LIN {X 0,Y 187.273,Z 370.418,A -85,B 0,C 180,E1 -25349.144,E2 -25349.144} C_VEL
LIN {X 0,Y 191.454,Z 356.11,A -85,B 0,C 180,E1 -25350.14,E2 -25350.14} C_VEL
LIN {X 0,Y 194.75,Z 340.819,A -85,B 0,C 180,E1 -25350.906,E2 -25350.906} C_VEL
LIN {X 0,Y 196.826,Z 325.628,A -85,B 0,C 180,E1 -25351.428,E2 -25351.428} C_VEL
LIN {X 0,Y 201.138,Z 277.904,A -85,B 0,C 180,E1 -25352.703,E2 -25352.703} C_VEL
LIN {X 0,Y 197.64,Z 268.624,A -85,B 0,C 180,E1 -25355.513,E2 -25355.513} C_VEL
LIN {X 0,Y 193.851,Z 261.276,A -85,B 0,C 180,E1 -25358.813,E2 -25358.813} C_VEL
LIN {X 0,Y 190.051,Z 254.613,A -85,B 0,C 180,E1 -25362.793,E2 -25362.793} C_VEL
LIN {X 0,Y 187.566,Z 250.534,A -85,B 0,C 180,E1 -25366.042,E2 -25366.042} C_VEL
LIN {X 0,Y 185.493,Z 246.833,A -85,B 0,C 180,E1 -25369.632,E2 -25369.632} C_VEL
LIN {X 0,Y 183.537,Z 243.434,A -85,B 0,C 180,E1 -25375.058,E2 -25375.058} C_VEL
LIN {X 0,Y 183.272,Z 242.439,A -85,B 0,C 180,E1 -25376.703,E2 -25376.703} C_VEL
LIN {X 0,Y 183.007,Z 241.999,A -85,B 0,C 180,E1 -25380,E2 -25380} C_VEL
LIN {X 0,Y 183.335,Z 242.534,A -85,B 0,C 180,E1 -25383.847,E2 -25383.847} C_VEL
LIN {X 0,Y 184.872,Z 246.218,A -85,B 0,C 180,E1 -25389.298,E2 -25389.298} C_VEL
LIN {X 0,Y 185.731,Z 247.38,A -85,B 0,C 180,E1 -25391.044,E2 -25391.044} C_VEL
LIN {X 0,Y 188.365,Z 251.957,A -85,B 0,C 180,E1 -25395.278,E2 -25395.278} C_VEL
LIN {X 0,Y 190.886,Z 256.242,A -85,B 0,C 180,E1 -25398.364,E2 -25398.364} C_VEL
LIN {X 0,Y 193.99,Z 261.588,A -85,B 0,C 180,E1 -25401.5,E2 -25401.5} C_VEL
LIN {X 0,Y 198.275,Z 269.947,A -85,B 0,C 180,E1 -25405.173,E2 -25405.173} C_VEL
LIN {X 0,Y 201.262,Z 276.327,A -85,B 0,C 180,E1 -25407.421,E2 -25407.421} C_VEL
LIN {X 0,Y 196.205,Z 330.798,A -85,B 0,C 180,E1 -25408.917,E2 -25408.917} C_VEL
LIN {X 0,Y 193.603,Z 345.867,A -85,B 0,C 180,E1 -25409.531,E2 -25409.531} C_VEL
LIN {X 0,Y 189.657,Z 361.736,A -85,B 0,C 180,E1 -25410.507,E2 -25410.507} C_VEL
LIN {X 0,Y 185.585,Z 374.397,A -85,B 0,C 180,E1 -25411.563,E2 -25411.563} C_VEL
LIN {X 0,Y 180.029,Z 388.733,A -85,B 0,C 180,E1 -25413.184,E2 -25413.184} C_VEL
LIN {X 0,Y 173.921,Z 401.727,A -85,B 0,C 180,E1 -25415.087,E2 -25415.087} C_VEL
LIN {X 0,Y 167.017,Z 414.16,A -85,B 0,C 180,E1 -25417.415,E2 -25417.415} C_VEL
LIN {X 0,Y 160.472,Z 424.572,A -85,B 0,C 180,E1 -25419.966,E2 -25419.966} C_VEL
LIN {X 0,Y 153.641,Z 434.234,A -85,B 0,C 180,E1 -25422.955,E2 -25422.955} C_VEL
LIN {X 0,Y 147.458,Z 442.478,A -85,B 0,C 180,E1 -25426.284,E2 -25426.284} C_VEL
LIN {X 0,Y 140.675,Z 450.588,A -85,B 0,C 180,E1 -25430.433,E2 -25430.433} C_VEL
LIN {X 0,Y 134.787,Z 457.281,A -85,B 0,C 180,E1 -25435.001,E2 -25435.001} C_VEL
LIN {X 0,Y 129.035,Z 463.475,A -85,B 0,C 180,E1 -25440.647,E2 -25440.647} C_VEL
LIN {X 0,Y 124.739,Z 468.254,A -85,B 0,C 180,E1 -25446.772,E2 -25446.772} C_VEL
LIN {X 0,Y 121.613,Z 471.753,A -85,B 0,C 180,E1 -25453.205,E2 -25453.205} C_VEL
LIN {X 0,Y 119.848,Z 474.061,A -85,B 0,C 180,E1 -25459.868,E2 -25459.868} C_VEL
LIN {X 0,Y 119.226,Z 475.233,A -85,B 0,C 180,E1 -25466.621,E2 -25466.621} C_VEL
LIN {X 0,Y 119.279,Z 475.389,A -85,B 0,C 180,E1 -25470,E2 -25470} C_VEL
LIN {X 0,Y 119.418,Z 474.819,A -85,B 0,C 180,E1 -25476.76,E2 -25476.76} C_VEL
LIN {X 0,Y 120.528,Z 473.127,A -85,B 0,C 180,E1 -25483.488,E2 -25483.488} C_VEL
LIN {X 0,Y 122.917,Z 470.27,A -85,B 0,C 180,E1 -25490.064,E2 -25490.064} C_VEL
LIN {X 0,Y 126.72,Z 466.181,A -85,B 0,C 180,E1 -25496.34,E2 -25496.34} C_VEL
LIN {X 0,Y 131.734,Z 460.761,A -85,B 0,C 180,E1 -25502.242,E2 -25502.242} C_VEL
LIN {X 0,Y 138.001,Z 453.855,A -85,B 0,C 180,E1 -25507.671,E2 -25507.671} C_VEL
LIN {X 0,Y 144.481,Z 446.434,A -85,B 0,C 180,E1 -25511.978,E2 -25511.978} C_VEL
LIN {X 0,Y 151.32,Z 437.625,A -85,B 0,C 180,E1 -25515.951,E2 -25515.951} C_VEL
LIN {X 0,Y 158.052,Z 428.371,A -85,B 0,C 180,E1 -25519.107,E2 -25519.107} C_VEL
LIN {X 0,Y 165.09,Z 417.612,A -85,B 0,C 180,E1 -25521.958,E2 -25521.958} C_VEL
LIN {X 0,Y 171.894,Z 405.866,A -85,B 0,C 180,E1 -25524.352,E2 -25524.352} C_VEL
LIN {X 0,Y 178.621,Z 392.289,A -85,B 0,C 180,E1 -25526.488,E2 -25526.488} C_VEL
LIN {X 0,Y 184.16,Z 378.874,A -85,B 0,C 180,E1 -25528.116,E2 -25528.116} C_VEL
LIN {X 0,Y 188.851,Z 365.062,A -85,B 0,C 180,E1 -25529.383,E2 -25529.383} C_VEL
LIN {X 0,Y 192.986,Z 349.593,A -85,B 0,C 180,E1 -25530.397,E2 -25530.397} C_VEL
LIN {X 0,Y 195.957,Z 333.83,A -85,B 0,C 180,E1 -25531.113,E2 -25531.113} C_VEL
LIN {X 0,Y 198.176,Z 313.58,A -85,B 0,C 180,E1 -25531.7,E2 -25531.7} C_VEL
LIN {X 0,Y 201.513,Z 276.593,A -85,B 0,C 180,E1 -25532.678,E2 -25532.678} C_VEL
LIN {X 0,Y 197.583,Z 268.293,A -85,B 0,C 180,E1 -25535.687,E2 -25535.687} C_VEL
LIN {X 0,Y 193.941,Z 261.297,A -85,B 0,C 180,E1 -25538.892,E2 -25538.892} C_VEL
LIN {X 0,Y 190.236,Z 254.787,A -85,B 0,C 180,E1 -25542.809,E2 -25542.809} C_VEL
LIN {X 0,Y 187.776,Z 250.724,A -85,B 0,C 180,E1 -25546.058,E2 -25546.058} C_VEL
LIN {X 0,Y 185.516,Z 246.776,A -85,B 0,C 180,E1 -25550.074,E2 -25550.074} C_VEL
LIN {X 0,Y 183.727,Z 243.503,A -85,B 0,C 180,E1 -25555.475,E2 -25555.475} C_VEL
LIN {X 0,Y 183.49,Z 242.512,A -85,B 0,C 180,E1 -25557.256,E2 -25557.256} C_VEL
LIN {X 0,Y 183.359,Z 242.216,A -85,B 0,C 180,E1 -25561.098,E2 -25561.098} C_VEL
LIN {X 0,Y 183.625,Z 242.95,A -85,B 0,C 180,E1 -25563.703,E2 -25563.703} C_VEL
LIN {X 0,Y 185.381,Z 246.651,A -85,B 0,C 180,E1 -25569.569,E2 -25569.569} C_VEL
LIN {X 0,Y 186.082,Z 247.75,A -85,B 0,C 180,E1 -25570.988,E2 -25570.988} C_VEL
LIN {X 0,Y 188.385,Z 251.662,A -85,B 0,C 180,E1 -25574.723,E2 -25574.723} C_VEL
LIN {X 0,Y 191.019,Z 256.175,A -85,B 0,C 180,E1 -25578.016,E2 -25578.016} C_VEL
LIN {X 0,Y 194.22,Z 261.783,A -85,B 0,C 180,E1 -25581.284,E2 -25581.284} C_VEL
LIN {X 0,Y 197.961,Z 269.051,A -85,B 0,C 180,E1 -25584.533,E2 -25584.533} C_VEL
LIN {X 0,Y 201.206,Z 277.645,A -85,B 0,C 180,E1 -25587.146,E2 -25587.146} C_VEL
LIN {X 0,Y 201.355,Z 278.122,A -85,B 0,C 180,E1 -25587.265,E2 -25587.265} C_VEL
LIN {X 0,Y 196.451,Z 331.048,A -85,B 0,C 180,E1 -25588.689,E2 -25588.689} C_VEL
LIN {X 0,Y 193.807,Z 346.99,A -85,B 0,C 180,E1 -25589.331,E2 -25589.331} C_VEL
LIN {X 0,Y 190.094,Z 362.089,A -85,B 0,C 180,E1 -25590.208,E2 -25590.208} C_VEL
LIN {X 0,Y 185.251,Z 376.98,A -85,B 0,C 180,E1 -25591.394,E2 -25591.394} C_VEL
LIN {X 0,Y 179.931,Z 390.407,A -85,B 0,C 180,E1 -25592.883,E2 -25592.883} C_VEL
LIN {X 0,Y 174.116,Z 402.855,A -85,B 0,C 180,E1 -25594.698,E2 -25594.698} C_VEL
LIN {X 0,Y 167.162,Z 415.39,A -85,B 0,C 180,E1 -25596.982,E2 -25596.982} C_VEL
LIN {X 0,Y 159.927,Z 426.838,A -85,B 0,C 180,E1 -25599.732,E2 -25599.732} C_VEL
LIN {X 0,Y 153.096,Z 436.472,A -85,B 0,C 180,E1 -25602.735,E2 -25602.735} C_VEL
LIN {X 0,Y 145.853,Z 445.912,A -85,B 0,C 180,E1 -25606.615,E2 -25606.615} C_VEL
LIN {X 0,Y 139.248,Z 453.822,A -85,B 0,C 180,E1 -25610.884,E2 -25610.884} C_VEL
LIN {X 0,Y 132.657,Z 461.182,A -85,B 0,C 180,E1 -25616.201,E2 -25616.201} C_VEL
LIN {X 0,Y 127.44,Z 466.938,A -85,B 0,C 180,E1 -25621.927,E2 -25621.927} C_VEL
LIN {X 0,Y 126.164,Z 468.36,A -85,B 0,C 180,E1 -25623.679,E2 -25623.679} C_VEL
LIN {X 0,Y 123.936,Z 470.161,A -85,B 0,C 180,E1 -25626.051,E2 -25626.051} C_VEL
LIN {X 0,Y 118.949,Z 472.706,A -85,B 0,C 180,E1 -25629.915,E2 -25629.915} C_VEL
LIN {X 0,Y 115.172,Z 474.35,A -85,B 0,C 180,E1 -25633.249,E2 -25633.249} C_VEL
LIN {X 0,Y 113.313,Z 475.355,A -85,B 0,C 180,E1 -25636.027,E2 -25636.027} C_VEL
LIN {X 0,Y 113.003,Z 475.62,A -85,B 0,C 180,E1 -25637.003,E2 -25637.003} C_VEL
LIN {X 0,Y 112.218,Z 476.962,A -85,B 0,C 180,E1 -25642.804,E2 -25642.804} C_VEL
LIN {X 0,Y 112.133,Z 477.552,A -85,B 0,C 180,E1 -25650,E2 -25650} C_VEL
LIN {X 0,Y 112.218,Z 476.942,A -85,B 0,C 180,E1 -25657.195,E2 -25657.195} C_VEL
LIN {X 0,Y 113.33,Z 475.188,A -85,B 0,C 180,E1 -25664.362,E2 -25664.362} C_VEL
LIN {X 0,Y 115.86,Z 472.268,A -85,B 0,C 180,E1 -25671.343,E2 -25671.343} C_VEL
LIN {X 0,Y 119.857,Z 468.113,A -85,B 0,C 180,E1 -25677.975,E2 -25677.975} C_VEL
LIN {X 0,Y 125.196,Z 462.613,A -85,B 0,C 180,E1 -25684.15,E2 -25684.15} C_VEL
LIN {X 0,Y 131.859,Z 455.619,A -85,B 0,C 180,E1 -25689.762,E2 -25689.762} C_VEL
LIN {X 0,Y 138.605,Z 448.139,A -85,B 0,C 180,E1 -25694.202,E2 -25694.202} C_VEL
LIN {X 0,Y 144.94,Z 440.474,A -85,B 0,C 180,E1 -25697.685,E2 -25697.685} C_VEL
LIN {X 0,Y 153.057,Z 429.911,A -85,B 0,C 180,E1 -25701.315,E2 -25701.315} C_VEL
LIN {X 0,Y 160.402,Z 419.061,A -85,B 0,C 180,E1 -25704.152,E2 -25704.152} C_VEL
LIN {X 0,Y 167.539,Z 407.215,A -85,B 0,C 180,E1 -25706.483,E2 -25706.483} C_VEL
LIN {X 0,Y 174.157,Z 394.252,A -85,B 0,C 180,E1 -25708.483,E2 -25708.483} C_VEL
LIN {X 0,Y 179.564,Z 381.685,A -85,B 0,C 180,E1 -25709.992,E2 -25709.992} C_VEL
LIN {X 0,Y 184.449,Z 368.164,A -85,B 0,C 180,E1 -25711.207,E2 -25711.207} C_VEL
LIN {X 0,Y 188.715,Z 353.175,A -85,B 0,C 180,E1 -25712.188,E2 -25712.188} C_VEL
LIN {X 0,Y 191.814,Z 338.464,A -85,B 0,C 180,E1 -25712.842,E2 -25712.842} C_VEL
LIN {X 0,Y 193.807,Z 322.736,A -85,B 0,C 180,E1 -25713.357,E2 -25713.357} C_VEL
LIN {X 0,Y 197.7,Z 281.128,A -85,B 0,C 180,E1 -25714.428,E2 -25714.428} C_VEL
LIN {X 0,Y 195.226,Z 274.198,A -85,B 0,C 180,E1 -25716.602,E2 -25716.602} C_VEL
LIN {X 0,Y 191.961,Z 267.52,A -85,B 0,C 180,E1 -25719.647,E2 -25719.647} C_VEL
LIN {X 0,Y 188.406,Z 261.007,A -85,B 0,C 180,E1 -25723.615,E2 -25723.615} C_VEL
LIN {X 0,Y 186.333,Z 257.36,A -85,B 0,C 180,E1 -25726.504,E2 -25726.504} C_VEL
LIN {X 0,Y 184.22,Z 253.547,A -85,B 0,C 180,E1 -25730.392,E2 -25730.392} C_VEL
LIN {X 0,Y 182.515,Z 250.047,A -85,B 0,C 180,E1 -25735.86,E2 -25735.86} C_VEL
LIN {X 0,Y 182.327,Z 249.369,A -85,B 0,C 180,E1 -25737.239,E2 -25737.239} C_VEL
LIN {X 0,Y 182.141,Z 249.049,A -85,B 0,C 180,E1 -25740,E2 -25740} C_VEL
LIN {X 0,Y 182.422,Z 249.536,A -85,B 0,C 180,E1 -25743.59,E2 -25743.59} C_VEL
LIN {X 0,Y 183.885,Z 253.211,A -85,B 0,C 180,E1 -25749.071,E2 -25749.071} C_VEL
LIN {X 0,Y 184.576,Z 254.245,A -85,B 0,C 180,E1 -25750.559,E2 -25750.559} C_VEL
LIN {X 0,Y 186.869,Z 258.42,A -85,B 0,C 180,E1 -25754.498,E2 -25754.498} C_VEL
LIN {X 0,Y 189.38,Z 262.933,A -85,B 0,C 180,E1 -25757.767,E2 -25757.767} C_VEL
LIN {X 0,Y 192.2,Z 268.115,A -85,B 0,C 180,E1 -25760.782,E2 -25760.782} C_VEL
LIN {X 0,Y 195.833,Z 275.481,A -85,B 0,C 180,E1 -25764.093,E2 -25764.093} C_VEL
LIN {X 0,Y 197.75,Z 279.713,A -85,B 0,C 180,E1 -25765.663,E2 -25765.663} C_VEL
LIN {X 0,Y 192.842,Z 331.138,A -85,B 0,C 180,E1 -25767.086,E2 -25767.086} C_VEL
LIN {X 0,Y 190.208,Z 345.944,A -85,B 0,C 180,E1 -25767.672,E2 -25767.672} C_VEL
LIN {X 0,Y 186.16,Z 361.81,A -85,B 0,C 180,E1 -25768.628,E2 -25768.628} C_VEL
LIN {X 0,Y 181.974,Z 374.469,A -85,B 0,C 180,E1 -25769.661,E2 -25769.661} C_VEL
LIN {X 0,Y 176.295,Z 388.619,A -85,B 0,C 180,E1 -25771.215,E2 -25771.215} C_VEL
LIN {X 0,Y 169.939,Z 401.797,A -85,B 0,C 180,E1 -25773.127,E2 -25773.127} C_VEL
LIN {X 0,Y 162.774,Z 414.23,A -85,B 0,C 180,E1 -25775.417,E2 -25775.417} C_VEL
LIN {X 0,Y 155.993,Z 424.641,A -85,B 0,C 180,E1 -25777.961,E2 -25777.961} C_VEL
LIN {X 0,Y 148.865,Z 434.303,A -85,B 0,C 180,E1 -25780.943,E2 -25780.943} C_VEL
LIN {X 0,Y 142.373,Z 442.547,A -85,B 0,C 180,E1 -25784.294,E2 -25784.294} C_VEL
LIN {X 0,Y 135.247,Z 450.656,A -85,B 0,C 180,E1 -25788.506,E2 -25788.506} C_VEL
LIN {X 0,Y 128.995,Z 457.349,A -85,B 0,C 180,E1 -25793.179,E2 -25793.179} C_VEL
LIN {X 0,Y 122.62,Z 463.795,A -85,B 0,C 180,E1 -25799.287,E2 -25799.287} C_VEL
LIN {X 0,Y 118.21,Z 468.322,A -85,B 0,C 180,E1 -25805.407,E2 -25805.407} C_VEL
LIN {X 0,Y 114.781,Z 471.82,A -85,B 0,C 180,E1 -25812.173,E2 -25812.173} C_VEL
LIN {X 0,Y 112.832,Z 474.128,A -85,B 0,C 180,E1 -25819.23,E2 -25819.23} C_VEL
LIN {X 0,Y 112.135,Z 475.3,A -85,B 0,C 180,E1 -25826.407,E2 -25826.407} C_VEL
LIN {X 0,Y 112.199,Z 475.455,A -85,B 0,C 180,E1 -25830,E2 -25830} C_VEL
LIN {X 0,Y 112.344,Z 474.886,A -85,B 0,C 180,E1 -25837.188,E2 -25837.188} C_VEL
LIN {X 0,Y 113.614,Z 473.193,A -85,B 0,C 180,E1 -25844.326,E2 -25844.326} C_VEL
LIN {X 0,Y 116.241,Z 470.336,A -85,B 0,C 180,E1 -25851.27,E2 -25851.27} C_VEL
LIN {X 0,Y 120.364,Z 466.246,A -85,B 0,C 180,E1 -25857.848,E2 -25857.848} C_VEL
LIN {X 0,Y 125.74,Z 460.826,A -85,B 0,C 180,E1 -25863.982,E2 -25863.982} C_VEL
LIN {X 0,Y 132.42,Z 453.92,A -85,B 0,C 180,E1 -25869.56,E2 -25869.56} C_VEL
LIN {X 0,Y 139.245,Z 446.499,A -85,B 0,C 180,E1 -25873.947,E2 -25873.947} C_VEL
LIN {X 0,Y 146.555,Z 437.559,A -85,B 0,C 180,E1 -25878.012,E2 -25878.012} C_VEL
LIN {X 0,Y 153.483,Z 428.434,A -85,B 0,C 180,E1 -25881.118,E2 -25881.118} C_VEL
LIN {X 0,Y 160.798,Z 417.675,A -85,B 0,C 180,E1 -25883.958,E2 -25883.958} C_VEL
LIN {X 0,Y 167.857,Z 405.929,A -85,B 0,C 180,E1 -25886.32,E2 -25886.32} C_VEL
LIN {X 0,Y 174.394,Z 393.2,A -85,B 0,C 180,E1 -25888.318,E2 -25888.318} C_VEL
LIN {X 0,Y 180.502,Z 378.935,A -85,B 0,C 180,E1 -25890.035,E2 -25890.035} C_VEL
LIN {X 0,Y 185.342,Z 365.121,A -85,B 0,C 180,E1 -25891.269,E2 -25891.269} C_VEL
LIN {X 0,Y 189.588,Z 349.649,A -85,B 0,C 180,E1 -25892.257,E2 -25892.257} C_VEL
LIN {X 0,Y 192.625,Z 333.903,A -85,B 0,C 180,E1 -25892.961,E2 -25892.961} C_VEL
LIN {X 0,Y 194.914,Z 313.624,A -85,B 0,C 180,E1 -25893.536,E2 -25893.536} C_VEL
LIN {X 0,Y 198.014,Z 279.985,A -85,B 0,C 180,E1 -25894.431,E2 -25894.431} C_VEL
LIN {X 0,Y 194.402,Z 272.251,A -85,B 0,C 180,E1 -25897.481,E2 -25897.481} C_VEL
LIN {X 0,Y 191.561,Z 266.693,A -85,B 0,C 180,E1 -25900.229,E2 -25900.229} C_VEL
LIN {X 0,Y 188.596,Z 261.203,A -85,B 0,C 180,E1 -25903.631,E2 -25903.631} C_VEL
LIN {X 0,Y 186.366,Z 257.303,A -85,B 0,C 180,E1 -25906.795,E2 -25906.795} C_VEL
LIN {X 0,Y 184.468,Z 253.72,A -85,B 0,C 180,E1 -25910.405,E2 -25910.405} C_VEL
LIN {X 0,Y 182.761,Z 250.331,A -85,B 0,C 180,E1 -25916.003,E2 -25916.003} C_VEL
LIN {X 0,Y 182.624,Z 249.578,A -85,B 0,C 180,E1 -25917.243,E2 -25917.243} C_VEL
LIN {X 0,Y 182.493,Z 249.271,A -85,B 0,C 180,E1 -25921.103,E2 -25921.103} C_VEL
LIN {X 0,Y 182.694,Z 249.88,A -85,B 0,C 180,E1 -25923.308,E2 -25923.308} C_VEL
LIN {X 0,Y 184.379,Z 253.633,A -85,B 0,C 180,E1 -25929.323,E2 -25929.323} C_VEL
LIN {X 0,Y 184.88,Z 254.489,A -85,B 0,C 180,E1 -25930.402,E2 -25930.402} C_VEL
LIN {X 0,Y 187.035,Z 258.4,A -85,B 0,C 180,E1 -25934.137,E2 -25934.137} C_VEL
LIN {X 0,Y 189.475,Z 262.8,A -85,B 0,C 180,E1 -25937.366,E2 -25937.366} C_VEL
LIN {X 0,Y 192.384,Z 268.166,A -85,B 0,C 180,E1 -25940.512,E2 -25940.512} C_VEL
LIN {X 0,Y 195.683,Z 274.907,A -85,B 0,C 180,E1 -25943.562,E2 -25943.562} C_VEL
LIN {X 0,Y 197.937,Z 281.292,A -85,B 0,C 180,E1 -25945.544,E2 -25945.544} C_VEL
LIN {X 0,Y 192.964,Z 332.343,A -85,B 0,C 180,E1 -25946.879,E2 -25946.879} C_VEL
LIN {X 0,Y 190.212,Z 348.008,A -85,B 0,C 180,E1 -25947.531,E2 -25947.531} C_VEL
LIN {X 0,Y 186.269,Z 363.213,A -85,B 0,C 180,E1 -25948.406,E2 -25948.406} C_VEL
LIN {X 0,Y 181.659,Z 376.919,A -85,B 0,C 180,E1 -25949.485,E2 -25949.485} C_VEL
LIN {X 0,Y 176.166,Z 390.346,A -85,B 0,C 180,E1 -25950.938,E2 -25950.938} C_VEL
LIN {X 0,Y 169.94,Z 403.229,A -85,B 0,C 180,E1 -25952.794,E2 -25952.794} C_VEL
LIN {X 0,Y 162.331,Z 416.396,A -85,B 0,C 180,E1 -25955.196,E2 -25955.196} C_VEL
LIN {X 0,Y 154.244,Z 428.529,A -85,B 0,C 180,E1 -25958.188,E2 -25958.188} C_VEL
LIN {X 0,Y 146.078,Z 439.323,A -85,B 0,C 180,E1 -25961.778,E2 -25961.778} C_VEL
LIN {X 0,Y 138.666,Z 448.316,A -85,B 0,C 180,E1 -25965.822,E2 -25965.822} C_VEL
LIN {X 0,Y 131.863,Z 455.776,A -85,B 0,C 180,E1 -25970.24,E2 -25970.24} C_VEL
LIN {X 0,Y 125.204,Z 462.732,A -85,B 0,C 180,E1 -25975.852,E2 -25975.852} C_VEL
LIN {X 0,Y 119.46,Z 468.625,A -85,B 0,C 180,E1 -25982.621,E2 -25982.621} C_VEL
LIN {X 0,Y 115.898,Z 472.336,A -85,B 0,C 180,E1 -25988.664,E2 -25988.664} C_VEL
LIN {X 0,Y 113.334,Z 475.234,A -85,B 0,C 180,E1 -25995.638,E2 -25995.638} C_VEL
LIN {X 0,Y 113.003,Z 475.62,A -85,B 0,C 180,E1 -25997.003,E2 -25997.003} C_VEL
LIN {X 0,Y 111.819,Z 476.422,A -85,B 0,C 180,E1 -25999.927,E2 -25999.927} C_VEL
LIN {X 0,Y 108.525,Z 477.215,A -85,B 0,C 180,E1 -26004.772,E2 -26004.772} C_VEL
LIN {X 0,Y 105.21,Z 477.45,A -85,B 0,C 180,E1 -26010.972,E2 -26010.972} C_VEL
LIN {X 0,Y 104.936,Z 477.355,A -85,B 0,C 180,E1 -26013.146,E2 -26013.146} C_VEL
LIN {X 0,Y 105.154,Z 476.875,A -85,B 0,C 180,E1 -26017.682,E2 -26017.682} C_VEL
LIN {X 0,Y 106.422,Z 475.12,A -85,B 0,C 180,E1 -26025.317,E2 -26025.317} C_VEL
LIN {X 0,Y 109.226,Z 472.2,A -85,B 0,C 180,E1 -26032.71,E2 -26032.71} C_VEL
LIN {X 0,Y 113.557,Z 468.045,A -85,B 0,C 180,E1 -26039.677,E2 -26039.677} C_VEL
LIN {X 0,Y 119.326,Z 462.545,A -85,B 0,C 180,E1 -26046.084,E2 -26046.084} C_VEL
LIN {X 0,Y 126.45,Z 455.55,A -85,B 0,C 180,E1 -26051.832,E2 -26051.832} C_VEL
LIN {X 0,Y 132.539,Z 449.194,A -85,B 0,C 180,E1 -26055.713,E2 -26055.713} C_VEL
LIN {X 0,Y 139.058,Z 441.761,A -85,B 0,C 180,E1 -26059.297,E2 -26059.297} C_VEL
LIN {X 0,Y 147.45,Z 431.472,A -85,B 0,C 180,E1 -26062.974,E2 -26062.974} C_VEL
LIN {X 0,Y 155.025,Z 420.944,A -85,B 0,C 180,E1 -26065.828,E2 -26065.828} C_VEL
LIN {X 0,Y 162.358,Z 409.494,A -85,B 0,C 180,E1 -26068.158,E2 -26068.158} C_VEL
LIN {X 0,Y 169.137,Z 397.071,A -85,B 0,C 180,E1 -26070.144,E2 -26070.144} C_VEL
LIN {X 0,Y 175.411,Z 383.38,A -85,B 0,C 180,E1 -26071.818,E2 -26071.818} C_VEL
LIN {X 0,Y 180.778,Z 369.219,A -85,B 0,C 180,E1 -26073.092,E2 -26073.092} C_VEL
LIN {X 0,Y 185.324,Z 353.861,A -85,B 0,C 180,E1 -26074.09,E2 -26074.09} C_VEL
LIN {X 0,Y 188.705,Z 338.262,A -85,B 0,C 180,E1 -26074.76,E2 -26074.76} C_VEL
LIN {X 0,Y 190.763,Z 322.35,A -85,B 0,C 180,E1 -26075.267,E2 -26075.267} C_VEL
LIN {X 0,Y 194.441,Z 284.269,A -85,B 0,C 180,E1 -26076.223,E2 -26076.223} C_VEL
LIN {X 0,Y 192.609,Z 279.087,A -85,B 0,C 180,E1 -26077.984,E2 -26077.984} C_VEL
LIN {X 0,Y 189.629,Z 272.915,A -85,B 0,C 180,E1 -26081.007,E2 -26081.007} C_VEL
LIN {X 0,Y 186.806,Z 267.362,A -85,B 0,C 180,E1 -26084.452,E2 -26084.452} C_VEL
LIN {X 0,Y 184.859,Z 263.835,A -85,B 0,C 180,E1 -26087.373,E2 -26087.373} C_VEL
LIN {X 0,Y 183.166,Z 260.451,A -85,B 0,C 180,E1 -26090.754,E2 -26090.754} C_VEL
LIN {X 0,Y 181.572,Z 256.99,A -85,B 0,C 180,E1 -26096.255,E2 -26096.255} C_VEL
LIN {X 0,Y 181.395,Z 256.324,A -85,B 0,C 180,E1 -26097.78,E2 -26097.78} C_VEL
LIN {X 0,Y 181.276,Z 256.098,A -85,B 0,C 180,E1 -26100,E2 -26100} C_VEL
LIN {X 0,Y 181.523,Z 256.657,A -85,B 0,C 180,E1 -26103.468,E2 -26103.468} C_VEL
LIN {X 0,Y 182.903,Z 260.193,A -85,B 0,C 180,E1 -26108.842,E2 -26108.842} C_VEL
LIN {X 0,Y 183.496,Z 261.239,A -85,B 0,C 180,E1 -26110.203,E2 -26110.203} C_VEL
LIN {X 0,Y 185.576,Z 265.224,A -85,B 0,C 180,E1 -26113.971,E2 -26113.971} C_VEL
LIN {X 0,Y 187.82,Z 269.478,A -85,B 0,C 180,E1 -26117.068,E2 -26117.068} C_VEL
LIN {X 0,Y 190.368,Z 274.434,A -85,B 0,C 180,E1 -26119.968,E2 -26119.968} C_VEL
LIN {X 0,Y 193.612,Z 281.408,A -85,B 0,C 180,E1 -26123.128,E2 -26123.128} C_VEL
LIN {X 0,Y 194.481,Z 283.403,A -85,B 0,C 180,E1 -26123.902,E2 -26123.902} C_VEL
LIN {X 0,Y 189.692,Z 331.384,A -85,B 0,C 180,E1 -26125.185,E2 -26125.185} C_VEL
LIN {X 0,Y 187.022,Z 346.021,A -85,B 0,C 180,E1 -26125.748,E2 -26125.748} C_VEL
LIN {X 0,Y 182.86,Z 361.883,A -85,B 0,C 180,E1 -26126.673,E2 -26126.673} C_VEL
LIN {X 0,Y 177.859,Z 376.402,A -85,B 0,C 180,E1 -26127.855,E2 -26127.855} C_VEL
LIN {X 0,Y 172.353,Z 389.504,A -85,B 0,C 180,E1 -26129.296,E2 -26129.296} C_VEL
LIN {X 0,Y 165.483,Z 403.108,A -85,B 0,C 180,E1 -26131.273,E2 -26131.273} C_VEL
LIN {X 0,Y 158.115,Z 415.336,A -85,B 0,C 180,E1 -26133.549,E2 -26133.549} C_VEL
LIN {X 0,Y 150.45,Z 426.481,A -85,B 0,C 180,E1 -26136.312,E2 -26136.312} C_VEL
LIN {X 0,Y 143.115,Z 435.856,A -85,B 0,C 180,E1 -26139.337,E2 -26139.337} C_VEL
LIN {X 0,Y 136.392,Z 443.843,A -85,B 0,C 180,E1 -26142.754,E2 -26142.754} C_VEL
LIN {X 0,Y 128.977,Z 451.73,A -85,B 0,C 180,E1 -26147.068,E2 -26147.068} C_VEL
LIN {X 0,Y 121.595,Z 459.092,A -85,B 0,C 180,E1 -26152.635,E2 -26152.635} C_VEL
LIN {X 0,Y 116.147,Z 464.227,A -85,B 0,C 180,E1 -26157.902,E2 -26157.902} C_VEL
LIN {X 0,Y 111.753,Z 468.389,A -85,B 0,C 180,E1 -26163.882,E2 -26163.882} C_VEL
LIN {X 0,Y 107.993,Z 471.888,A -85,B 0,C 180,E1 -26171.011,E2 -26171.011} C_VEL
LIN {X 0,Y 105.845,Z 474.195,A -85,B 0,C 180,E1 -26178.51,E2 -26178.51} C_VEL
LIN {X 0,Y 105.045,Z 475.366,A -85,B 0,C 180,E1 -26186.164,E2 -26186.164} C_VEL
LIN {X 0,Y 105.106,Z 475.521,A -85,B 0,C 180,E1 -26190,E2 -26190} C_VEL
LIN {X 0,Y 105.287,Z 474.952,A -85,B 0,C 180,E1 -26197.672,E2 -26197.672} C_VEL
LIN {X 0,Y 106.717,Z 473.259,A -85,B 0,C 180,E1 -26205.274,E2 -26205.274} C_VEL
LIN {X 0,Y 109.628,Z 470.402,A -85,B 0,C 180,E1 -26212.622,E2 -26212.622} C_VEL
LIN {X 0,Y 114.097,Z 466.312,A -85,B 0,C 180,E1 -26219.523,E2 -26219.523} C_VEL
LIN {X 0,Y 119.876,Z 460.892,A -85,B 0,C 180,E1 -26225.893,E2 -26225.893} C_VEL
LIN {X 0,Y 126.987,Z 453.985,A -85,B 0,C 180,E1 -26231.616,E2 -26231.616} C_VEL
LIN {X 0,Y 135.236,Z 445.365,A -85,B 0,C 180,E1 -26236.682,E2 -26236.682} C_VEL
LIN {X 0,Y 142.928,Z 436.352,A -85,B 0,C 180,E1 -26240.645,E2 -26240.645} C_VEL
LIN {X 0,Y 150.373,Z 426.874,A -85,B 0,C 180,E1 -26243.728,E2 -26243.728} C_VEL
LIN {X 0,Y 158.026,Z 415.789,A -85,B 0,C 180,E1 -26246.5,E2 -26246.5} C_VEL
LIN {X 0,Y 165.376,Z 403.647,A -85,B 0,C 180,E1 -26248.788,E2 -26248.788} C_VEL
LIN {X 0,Y 172.192,Z 390.32,A -85,B 0,C 180,E1 -26250.739,E2 -26250.739} C_VEL
LIN {X 0,Y 177.76,Z 377.231,A -85,B 0,C 180,E1 -26252.206,E2 -26252.206} C_VEL
LIN {X 0,Y 182.423,Z 364.05,A -85,B 0,C 180,E1 -26253.294,E2 -26253.294} C_VEL
LIN {X 0,Y 186.576,Z 348.944,A -85,B 0,C 180,E1 -26254.225,E2 -26254.225} C_VEL
LIN {X 0,Y 189.451,Z 334.301,A -85,B 0,C 180,E1 -26254.859,E2 -26254.859} C_VEL
LIN {X 0,Y 191.799,Z 314.349,A -85,B 0,C 180,E1 -26255.411,E2 -26255.411} C_VEL
LIN {X 0,Y 194.684,Z 283.513,A -85,B 0,C 180,E1 -26256.247,E2 -26256.247} C_VEL
LIN {X 0,Y 191.136,Z 275.626,A -85,B 0,C 180,E1 -26259.619,E2 -26259.619} C_VEL
LIN {X 0,Y 188.177,Z 269.853,A -85,B 0,C 180,E1 -26262.93,E2 -26262.93} C_VEL
LIN {X 0,Y 185.413,Z 264.507,A -85,B 0,C 180,E1 -26266.854,E2 -26266.854} C_VEL
LIN {X 0,Y 183.324,Z 260.558,A -85,B 0,C 180,E1 -26270.965,E2 -26270.965} C_VEL
LIN {X 0,Y 181.786,Z 256.956,A -85,B 0,C 180,E1 -26276.814,E2 -26276.814} C_VEL
LIN {X 0,Y 181.619,Z 256.346,A -85,B 0,C 180,E1 -26278.891,E2 -26278.891} C_VEL
LIN {X 0,Y 181.627,Z 256.328,A -85,B 0,C 180,E1 -26281.108,E2 -26281.108} C_VEL
LIN {X 0,Y 181.794,Z 257.015,A -85,B 0,C 180,E1 -26283.185,E2 -26283.185} C_VEL
LIN {X 0,Y 183.635,Z 261.071,A -85,B 0,C 180,E1 -26289.661,E2 -26289.661} C_VEL
LIN {X 0,Y 185.768,Z 265.253,A -85,B 0,C 180,E1 -26293.642,E2 -26293.642} C_VEL
LIN {X 0,Y 187.902,Z 269.294,A -85,B 0,C 180,E1 -26296.634,E2 -26296.634} C_VEL
LIN {X 0,Y 190.42,Z 274.178,A -85,B 0,C 180,E1 -26299.546,E2 -26299.546} C_VEL
LIN {X 0,Y 193.388,Z 280.613,A -85,B 0,C 180,E1 -26302.502,E2 -26302.502} C_VEL
LIN {X 0,Y 194.683,Z 284.414,A -85,B 0,C 180,E1 -26303.746,E2 -26303.746} C_VEL
LIN {X 0,Y 189.841,Z 332.399,A -85,B 0,C 180,E1 -26304.97,E2 -26304.97} C_VEL
LIN {X 0,Y 187.031,Z 347.951,A -85,B 0,C 180,E1 -26305.599,E2 -26305.599} C_VEL
LIN {X 0,Y 183.003,Z 363.154,A -85,B 0,C 180,E1 -26306.454,E2 -26306.454} C_VEL
LIN {X 0,Y 178.269,Z 376.859,A -85,B 0,C 180,E1 -26307.497,E2 -26307.497} C_VEL
LIN {X 0,Y 172.613,Z 390.284,A -85,B 0,C 180,E1 -26308.91,E2 -26308.91} C_VEL
LIN {X 0,Y 165.949,Z 403.618,A -85,B 0,C 180,E1 -26310.797,E2 -26310.797} C_VEL
LIN {X 0,Y 158.344,Z 416.333,A -85,B 0,C 180,E1 -26313.096,E2 -26313.096} C_VEL
LIN {X 0,Y 149.938,Z 428.465,A -85,B 0,C 180,E1 -26316.045,E2 -26316.045} C_VEL
LIN {X 0,Y 141.418,Z 439.258,A -85,B 0,C 180,E1 -26319.619,E2 -26319.619} C_VEL
LIN {X 0,Y 133.61,Z 448.25,A -85,B 0,C 180,E1 -26323.675,E2 -26323.675} C_VEL
LIN {X 0,Y 126.453,Z 455.71,A -85,B 0,C 180,E1 -26328.169,E2 -26328.169} C_VEL
LIN {X 0,Y 119.333,Z 462.666,A -85,B 0,C 180,E1 -26333.918,E2 -26333.918} C_VEL
LIN {X 0,Y 113.585,Z 468.135,A -85,B 0,C 180,E1 -26340.33,E2 -26340.33} C_VEL
LIN {X 0,Y 109.26,Z 472.27,A -85,B 0,C 180,E1 -26347.298,E2 -26347.298} C_VEL
LIN {X 0,Y 106.428,Z 475.167,A -85,B 0,C 180,E1 -26354.684,E2 -26354.684} C_VEL
LIN {X 0,Y 105.154,Z 476.896,A -85,B 0,C 180,E1 -26362.318,E2 -26362.318} C_VEL
LIN {X 0,Y 105.033,Z 477.486,A -85,B 0,C 180,E1 -26370,E2 -26370} C_VEL
LIN {X 0,Y 104.936,Z 477.355,A -85,B 0,C 180,E1 -26373.146,E2 -26373.146} C_VEL
LIN {X 0,Y 104.69,Z 477.222,A -85,B 0,C 180,E1 -26375.292,E2 -26375.292} C_VEL
LIN {X 0,Y 103.563,Z 476.861,A -85,B 0,C 180,E1 -26378.49,E2 -26378.49} C_VEL
LIN {X 0,Y 100.56,Z 475.215,A -85,B 0,C 180,E1 -26386.106,E2 -26386.106} C_VEL
LIN {X 0,Y 100.562,Z 474.11,A -85,B 0,C 180,E1 -26389.444,E2 -26389.444} C_VEL
LIN {X 0,Y 100.902,Z 473.685,A -85,B 0,C 180,E1 -26390.531,E2 -26390.531} C_VEL
LIN {X 0,Y 104.856,Z 470.215,A -85,B 0,C 180,E1 -26397.981,E2 -26397.981} C_VEL
LIN {X 0,Y 110.293,Z 465.403,A -85,B 0,C 180,E1 -26404.994,E2 -26404.994} C_VEL
LIN {X 0,Y 117.28,Z 459.177,A -85,B 0,C 180,E1 -26411.237,E2 -26411.237} C_VEL
LIN {X 0,Y 125.51,Z 451.362,A -85,B 0,C 180,E1 -26416.714,E2 -26416.714} C_VEL
LIN {X 0,Y 131.952,Z 444.485,A -85,B 0,C 180,E1 -26420.393,E2 -26420.393} C_VEL
LIN {X 0,Y 140.717,Z 434.558,A -85,B 0,C 180,E1 -26424.252,E2 -26424.252} C_VEL
LIN {X 0,Y 148.459,Z 424.579,A -85,B 0,C 180,E1 -26427.17,E2 -26427.17} C_VEL
LIN {X 0,Y 155.939,Z 413.796,A -85,B 0,C 180,E1 -26429.536,E2 -26429.536} C_VEL
LIN {X 0,Y 163.071,Z 401.899,A -85,B 0,C 180,E1 -26431.566,E2 -26431.566} C_VEL
LIN {X 0,Y 169.283,Z 389.712,A -85,B 0,C 180,E1 -26433.202,E2 -26433.202} C_VEL
LIN {X 0,Y 175.078,Z 376.16,A -85,B 0,C 180,E1 -26434.581,E2 -26434.581} C_VEL
LIN {X 0,Y 180.286,Z 361.087,A -85,B 0,C 180,E1 -26435.674,E2 -26435.674} C_VEL
LIN {X 0,Y 184.222,Z 346.039,A -85,B 0,C 180,E1 -26436.443,E2 -26436.443} C_VEL
LIN {X 0,Y 186.966,Z 330.419,A -85,B 0,C 180,E1 -26437.013,E2 -26437.013} C_VEL
LIN {X 0,Y 191.349,Z 287.399,A -85,B 0,C 180,E1 -26438.101,E2 -26438.101} C_VEL
LIN {X 0,Y 189.809,Z 283.38,A -85,B 0,C 180,E1 -26439.706,E2 -26439.706} C_VEL
LIN {X 0,Y 186.896,Z 277.081,A -85,B 0,C 180,E1 -26443.057,E2 -26443.057} C_VEL
LIN {X 0,Y 184.875,Z 273.134,A -85,B 0,C 180,E1 -26445.835,E2 -26445.835} C_VEL
LIN {X 0,Y 183.469,Z 270.344,A -85,B 0,C 180,E1 -26448.188,E2 -26448.188} C_VEL
LIN {X 0,Y 182.115,Z 267.388,A -85,B 0,C 180,E1 -26451.12,E2 -26451.12} C_VEL
LIN {X 0,Y 180.626,Z 263.816,A -85,B 0,C 180,E1 -26456.794,E2 -26456.794} C_VEL
LIN {X 0,Y 180.437,Z 263.254,A -85,B 0,C 180,E1 -26458.884,E2 -26458.884} C_VEL
LIN {X 0,Y 180.602,Z 263.574,A -85,B 0,C 180,E1 -26463.067,E2 -26463.067} C_VEL
LIN {X 0,Y 181.866,Z 267.121,A -85,B 0,C 180,E1 -26468.472,E2 -26468.472} C_VEL
LIN {X 0,Y 182.421,Z 268.251,A -85,B 0,C 180,E1 -26469.844,E2 -26469.844} C_VEL
LIN {X 0,Y 184.279,Z 271.998,A -85,B 0,C 180,E1 -26473.407,E2 -26473.407} C_VEL
LIN {X 0,Y 186.196,Z 275.829,A -85,B 0,C 180,E1 -26476.234,E2 -26476.234} C_VEL
LIN {X 0,Y 188.475,Z 280.523,A -85,B 0,C 180,E1 -26479.023,E2 -26479.023} C_VEL
LIN {X 0,Y 191.357,Z 287.084,A -85,B 0,C 180,E1 -26482.05,E2 -26482.05} C_VEL
LIN {X 0,Y 186.799,Z 331.304,A -85,B 0,C 180,E1 -26483.202,E2 -26483.202} C_VEL
LIN {X 0,Y 184.043,Z 346.097,A -85,B 0,C 180,E1 -26483.753,E2 -26483.753} C_VEL
LIN {X 0,Y 179.782,Z 361.957,A -85,B 0,C 180,E1 -26484.648,E2 -26484.648} C_VEL
LIN {X 0,Y 174.66,Z 376.474,A -85,B 0,C 180,E1 -26485.798,E2 -26485.798} C_VEL
LIN {X 0,Y 168.585,Z 390.384,A -85,B 0,C 180,E1 -26487.295,E2 -26487.295} C_VEL
LIN {X 0,Y 161.911,Z 403.178,A -85,B 0,C 180,E1 -26489.125,E2 -26489.125} C_VEL
LIN {X 0,Y 154.286,Z 415.406,A -85,B 0,C 180,E1 -26491.34,E2 -26491.34} C_VEL
LIN {X 0,Y 146.349,Z 426.55,A -85,B 0,C 180,E1 -26494.067,E2 -26494.067} C_VEL
LIN {X 0,Y 137.475,Z 437.374,A -85,B 0,C 180,E1 -26497.593,E2 -26497.593} C_VEL
LIN {X 0,Y 129.397,Z 446.358,A -85,B 0,C 180,E1 -26501.685,E2 -26501.685} C_VEL
LIN {X 0,Y 121.781,Z 453.808,A -85,B 0,C 180,E1 -26506.17,E2 -26506.17} C_VEL
LIN {X 0,Y 114.214,Z 460.768,A -85,B 0,C 180,E1 -26512.024,E2 -26512.024} C_VEL
LIN {X 0,Y 107.921,Z 466.236,A -85,B 0,C 180,E1 -26518.602,E2 -26518.602} C_VEL
LIN {X 0,Y 103.114,Z 470.36,A -85,B 0,C 180,E1 -26525.861,E2 -26525.861} C_VEL
LIN {X 0,Y 99.894,Z 473.253,A -85,B 0,C 180,E1 -26533.655,E2 -26533.655} C_VEL
LIN {X 0,Y 98.258,Z 474.987,A -85,B 0,C 180,E1 -26541.776,E2 -26541.776} C_VEL
LIN {X 0,Y 98.006,Z 475.588,A -85,B 0,C 180,E1 -26550,E2 -26550} C_VEL
LIN {X 0,Y 98.254,Z 475.018,A -85,B 0,C 180,E1 -26558.225,E2 -26558.225} C_VEL
LIN {X 0,Y 99.837,Z 473.325,A -85,B 0,C 180,E1 -26566.355,E2 -26566.355} C_VEL
LIN {X 0,Y 103.086,Z 470.468,A -85,B 0,C 180,E1 -26574.146,E2 -26574.146} C_VEL
LIN {X 0,Y 107.935,Z 466.378,A -85,B 0,C 180,E1 -26581.393,E2 -26581.393} C_VEL
LIN {X 0,Y 114.158,Z 460.957,A -85,B 0,C 180,E1 -26587.999,E2 -26587.999} C_VEL
LIN {X 0,Y 121.716,Z 454.051,A -85,B 0,C 180,E1 -26593.86,E2 -26593.86} C_VEL
LIN {X 0,Y 129.312,Z 446.63,A -85,B 0,C 180,E1 -26598.358,E2 -26598.358} C_VEL
LIN {X 0,Y 136.202,Z 439.036,A -85,B 0,C 180,E1 -26601.897,E2 -26601.897} C_VEL
LIN {X 0,Y 144.958,Z 428.562,A -85,B 0,C 180,E1 -26605.509,E2 -26605.509} C_VEL
LIN {X 0,Y 152.852,Z 417.802,A -85,B 0,C 180,E1 -26608.279,E2 -26608.279} C_VEL
LIN {X 0,Y 160.418,Z 406.054,A -85,B 0,C 180,E1 -26610.544,E2 -26610.544} C_VEL
LIN {X 0,Y 167.73,Z 392.6,A -85,B 0,C 180,E1 -26612.554,E2 -26612.554} C_VEL
LIN {X 0,Y 173.843,Z 379.056,A -85,B 0,C 180,E1 -26614.094,E2 -26614.094} C_VEL
LIN {X 0,Y 178.965,Z 365.239,A -85,B 0,C 180,E1 -26615.248,E2 -26615.248} C_VEL
LIN {X 0,Y 183.423,Z 349.762,A -85,B 0,C 180,E1 -26616.177,E2 -26616.177} C_VEL
LIN {X 0,Y 186.437,Z 335.017,A -85,B 0,C 180,E1 -26616.811,E2 -26616.811} C_VEL
LIN {X 0,Y 188.766,Z 316.361,A -85,B 0,C 180,E1 -26617.316,E2 -26617.316} C_VEL
LIN {X 0,Y 191.607,Z 287.288,A -85,B 0,C 180,E1 -26618.064,E2 -26618.064} C_VEL
LIN {X 0,Y 188.485,Z 280.146,A -85,B 0,C 180,E1 -26621.381,E2 -26621.381} C_VEL
LIN {X 0,Y 185.643,Z 274.287,A -85,B 0,C 180,E1 -26625.038,E2 -26625.038} C_VEL
LIN {X 0,Y 183.658,Z 270.497,A -85,B 0,C 180,E1 -26628.27,E2 -26628.27} C_VEL
LIN {X 0,Y 182.37,Z 267.554,A -85,B 0,C 180,E1 -26631.132,E2 -26631.132} C_VEL
LIN {X 0,Y 180.89,Z 264.072,A -85,B 0,C 180,E1 -26636.937,E2 -26636.937} C_VEL
LIN {X 0,Y 180.832,Z 263.571,A -85,B 0,C 180,E1 -26637.772,E2 -26637.772} C_VEL
LIN {X 0,Y 180.76,Z 263.385,A -85,B 0,C 180,E1 -26641.114,E2 -26641.114} C_VEL
LIN {X 0,Y 180.88,Z 263.989,A -85,B 0,C 180,E1 -26642.853,E2 -26642.853} C_VEL
LIN {X 0,Y 182.558,Z 268.072,A -85,B 0,C 180,E1 -26649.277,E2 -26649.277} C_VEL
LIN {X 0,Y 184.398,Z 271.846,A -85,B 0,C 180,E1 -26652.939,E2 -26652.939} C_VEL
LIN {X 0,Y 186.607,Z 276.273,A -85,B 0,C 180,E1 -26656.218,E2 -26656.218} C_VEL
LIN {X 0,Y 189.418,Z 282.182,A -85,B 0,C 180,E1 -26659.581,E2 -26659.581} C_VEL
LIN {X 0,Y 191.413,Z 287.058,A -85,B 0,C 180,E1 -26661.682,E2 -26661.682} C_VEL
LIN {X 0,Y 191.596,Z 287.648,A -85,B 0,C 180,E1 -26661.877,E2 -26661.877} C_VEL
LIN {X 0,Y 186.997,Z 332.142,A -85,B 0,C 180,E1 -26662.997,E2 -26662.997} C_VEL
LIN {X 0,Y 184.072,Z 347.894,A -85,B 0,C 180,E1 -26663.603,E2 -26663.603} C_VEL
LIN {X 0,Y 179.944,Z 363.095,A -85,B 0,C 180,E1 -26664.424,E2 -26664.424} C_VEL
LIN {X 0,Y 175.097,Z 376.798,A -85,B 0,C 180,E1 -26665.431,E2 -26665.431} C_VEL
LIN {X 0,Y 169.298,Z 390.223,A -85,B 0,C 180,E1 -26666.808,E2 -26666.808} C_VEL
LIN {X 0,Y 162.492,Z 403.388,A -85,B 0,C 180,E1 -26668.602,E2 -26668.602} C_VEL
LIN {X 0,Y 154.575,Z 416.27,A -85,B 0,C 180,E1 -26670.886,E2 -26670.886} C_VEL
LIN {X 0,Y 147.175,Z 426.647,A -85,B 0,C 180,E1 -26673.314,E2 -26673.314} C_VEL
LIN {X 0,Y 139.435,Z 436.279,A -85,B 0,C 180,E1 -26676.249,E2 -26676.249} C_VEL
LIN {X 0,Y 131.623,Z 445.106,A -85,B 0,C 180,E1 -26679.847,E2 -26679.847} C_VEL
LIN {X 0,Y 123.379,Z 453.626,A -85,B 0,C 180,E1 -26684.599,E2 -26684.599} C_VEL
LIN {X 0,Y 115.42,Z 460.985,A -85,B 0,C 180,E1 -26690.256,E2 -26690.256} C_VEL
LIN {X 0,Y 108.694,Z 466.947,A -85,B 0,C 180,E1 -26696.882,E2 -26696.882} C_VEL
LIN {X 0,Y 104.873,Z 470.296,A -85,B 0,C 180,E1 -26702.024,E2 -26702.024} C_VEL
LIN {X 0,Y 100.864,Z 473.802,A -85,B 0,C 180,E1 -26709.611,E2 -26709.611} C_VEL
LIN {X 0,Y 98.632,Z 476.108,A -85,B 0,C 180,E1 -26717.657,E2 -26717.657} C_VEL
LIN {X 0,Y 97.883,Z 477.267,A -85,B 0,C 180,E1 -26725.882,E2 -26725.882} C_VEL
LIN {X 0,Y 97.94,Z 477.419,A -85,B 0,C 180,E1 -26730,E2 -26730} C_VEL
LIN {X 0,Y 98.094,Z 476.809,A -85,B 0,C 180,E1 -26738.238,E2 -26738.238} C_VEL
LIN {X 0,Y 99.556,Z 475.053,A -85,B 0,C 180,E1 -26746.402,E2 -26746.402} C_VEL
LIN {X 0,Y 100.902,Z 473.685,A -85,B 0,C 180,E1 -26750.531,E2 -26750.531} C_VEL
LIN {X 0,Y 101.685,Z 472.439,A -85,B 0,C 180,E1 -26753.763,E2 -26753.763} C_VEL
LIN {X 0,Y 101.827,Z 470.042,A -85,B 0,C 180,E1 -26759.201,E2 -26759.201} C_VEL
LIN {X 0,Y 102.385,Z 467.866,A -85,B 0,C 180,E1 -26763.492,E2 -26763.492} C_VEL
LIN {X 0,Y 103.874,Z 465.933,A -85,B 0,C 180,E1 -26766.49,E2 -26766.49} C_VEL
LIN {X 0,Y 104.667,Z 465.203,A -85,B 0,C 180,E1 -26767.403,E2 -26767.403} C_VEL
LIN {X 0,Y 111.981,Z 459.109,A -85,B 0,C 180,E1 -26773.659,E2 -26773.659} C_VEL
LIN {X 0,Y 120.704,Z 451.294,A -85,B 0,C 180,E1 -26779.194,E2 -26779.194} C_VEL
LIN {X 0,Y 127.69,Z 444.247,A -85,B 0,C 180,E1 -26782.944,E2 -26782.944} C_VEL
LIN {X 0,Y 136.676,Z 434.489,A -85,B 0,C 180,E1 -26786.677,E2 -26786.677} C_VEL
LIN {X 0,Y 144.713,Z 424.51,A -85,B 0,C 180,E1 -26789.545,E2 -26789.545} C_VEL
LIN {X 0,Y 153.166,Z 412.657,A -85,B 0,C 180,E1 -26792.041,E2 -26792.041} C_VEL
LIN {X 0,Y 159.788,Z 401.828,A -85,B 0,C 180,E1 -26793.822,E2 -26793.822} C_VEL
LIN {X 0,Y 166.196,Z 389.64,A -85,B 0,C 180,E1 -26795.392,E2 -26795.392} C_VEL
LIN {X 0,Y 172.156,Z 376.088,A -85,B 0,C 180,E1 -26796.712,E2 -26796.712} C_VEL
LIN {X 0,Y 177.096,Z 362.288,A -85,B 0,C 180,E1 -26797.691,E2 -26797.691} C_VEL
LIN {X 0,Y 181.323,Z 346.784,A -85,B 0,C 180,E1 -26798.471,E2 -26798.471} C_VEL
LIN {X 0,Y 184.212,Z 331.184,A -85,B 0,C 180,E1 -26799.017,E2 -26799.017} C_VEL
LIN {X 0,Y 188.336,Z 292.213,A -85,B 0,C 180,E1 -26799.967,E2 -26799.967} C_VEL
LIN {X 0,Y 188.371,Z 290.669,A -85,B 0,C 180,E1 -26800.105,E2 -26800.105} C_VEL
LIN {X 0,Y 185.957,Z 285.075,A -85,B 0,C 180,E1 -26802.969,E2 -26802.969} C_VEL
LIN {X 0,Y 183.634,Z 279.974,A -85,B 0,C 180,E1 -26806.302,E2 -26806.302} C_VEL
LIN {X 0,Y 182.257,Z 277.112,A -85,B 0,C 180,E1 -26808.743,E2 -26808.743} C_VEL
LIN {X 0,Y 180.903,Z 274.133,A -85,B 0,C 180,E1 -26811.904,E2 -26811.904} C_VEL
LIN {X 0,Y 179.662,Z 270.446,A -85,B 0,C 180,E1 -26817.758,E2 -26817.758} C_VEL
LIN {X 0,Y 179.562,Z 270.289,A -85,B 0,C 180,E1 -26821.122,E2 -26821.122} C_VEL
LIN {X 0,Y 179.714,Z 270.815,A -85,B 0,C 180,E1 -26823.083,E2 -26823.083} C_VEL
LIN {X 0,Y 180.918,Z 274.142,A -85,B 0,C 180,E1 -26828.306,E2 -26828.306} C_VEL
LIN {X 0,Y 182.871,Z 278.484,A -85,B 0,C 180,E1 -26832.603,E2 -26832.603} C_VEL
LIN {X 0,Y 184.942,Z 282.875,A -85,B 0,C 180,E1 -26835.851,E2 -26835.851} C_VEL
LIN {X 0,Y 187.465,Z 288.505,A -85,B 0,C 180,E1 -26839.046,E2 -26839.046} C_VEL
LIN {X 0,Y 188.436,Z 290.888,A -85,B 0,C 180,E1 -26840.149,E2 -26840.149} C_VEL
LIN {X 0,Y 184.139,Z 331.277,A -85,B 0,C 180,E1 -26841.17,E2 -26841.17} C_VEL
LIN {X 0,Y 181.296,Z 346.174,A -85,B 0,C 180,E1 -26841.696,E2 -26841.696} C_VEL
LIN {X 0,Y 176.942,Z 362.031,A -85,B 0,C 180,E1 -26842.561,E2 -26842.561} C_VEL
LIN {X 0,Y 171.692,Z 376.546,A -85,B 0,C 180,E1 -26843.667,E2 -26843.667} C_VEL
LIN {X 0,Y 165.572,Z 390.205,A -85,B 0,C 180,E1 -26845.074,E2 -26845.074} C_VEL
LIN {X 0,Y 158.575,Z 403.249,A -85,B 0,C 180,E1 -26846.882,E2 -26846.882} C_VEL
LIN {X 0,Y 150.715,Z 415.476,A -85,B 0,C 180,E1 -26849.034,E2 -26849.034} C_VEL
LIN {X 0,Y 142.48,Z 426.62,A -85,B 0,C 180,E1 -26851.693,E2 -26851.693} C_VEL
LIN {X 0,Y 134.523,Z 435.993,A -85,B 0,C 180,E1 -26854.63,E2 -26854.63} C_VEL
LIN {X 0,Y 127.078,Z 444.018,A -85,B 0,C 180,E1 -26858.032,E2 -26858.032} C_VEL
LIN {X 0,Y 118.93,Z 451.866,A -85,B 0,C 180,E1 -26862.382,E2 -26862.382} C_VEL
LIN {X 0,Y 110.572,Z 459.228,A -85,B 0,C 180,E1 -26868.135,E2 -26868.135} C_VEL
LIN {X 0,Y 103.492,Z 464.982,A -85,B 0,C 180,E1 -26874.578,E2 -26874.578} C_VEL
LIN {X 0,Y 99.077,Z 468.525,A -85,B 0,C 180,E1 -26880.229,E2 -26880.229} C_VEL
LIN {X 0,Y 94.586,Z 472.022,A -85,B 0,C 180,E1 -26888.191,E2 -26888.191} C_VEL
LIN {X 0,Y 91.928,Z 474.329,A -85,B 0,C 180,E1 -26896.741,E2 -26896.741} C_VEL
LIN {X 0,Y 90.882,Z 475.499,A -85,B 0,C 180,E1 -26905.565,E2 -26905.565} C_VEL
LIN {X 0,Y 90.913,Z 475.654,A -85,B 0,C 180,E1 -26910,E2 -26910} C_VEL
LIN {X 0,Y 91.221,Z 475.085,A -85,B 0,C 180,E1 -26918.864,E2 -26918.864} C_VEL
LIN {X 0,Y 93.005,Z 473.392,A -85,B 0,C 180,E1 -26927.594,E2 -26927.594} C_VEL
LIN {X 0,Y 96.626,Z 470.534,A -85,B 0,C 180,E1 -26935.875,E2 -26935.875} C_VEL
LIN {X 0,Y 101.905,Z 466.444,A -85,B 0,C 180,E1 -26943.486,E2 -26943.486} C_VEL
LIN {X 0,Y 108.626,Z 461.023,A -85,B 0,C 180,E1 -26950.315,E2 -26950.315} C_VEL
LIN {X 0,Y 116.654,Z 454.116,A -85,B 0,C 180,E1 -26956.3,E2 -26956.3} C_VEL
LIN {X 0,Y 124.678,Z 446.695,A -85,B 0,C 180,E1 -26960.812,E2 -26960.812} C_VEL
LIN {X 0,Y 133.179,Z 437.75,A -85,B 0,C 180,E1 -26964.881,E2 -26964.881} C_VEL
LIN {X 0,Y 141.053,Z 428.626,A -85,B 0,C 180,E1 -26967.891,E2 -26967.891} C_VEL
LIN {X 0,Y 149.239,Z 417.865,A -85,B 0,C 180,E1 -26970.599,E2 -26970.599} C_VEL
LIN {X 0,Y 157.042,Z 406.116,A -85,B 0,C 180,E1 -26972.805,E2 -26972.805} C_VEL
LIN {X 0,Y 164.181,Z 393.43,A -85,B 0,C 180,E1 -26974.655,E2 -26974.655} C_VEL
LIN {X 0,Y 170.857,Z 379.117,A -85,B 0,C 180,E1 -26976.239,E2 -26976.239} C_VEL
LIN {X 0,Y 176.118,Z 365.298,A -85,B 0,C 180,E1 -26977.341,E2 -26977.341} C_VEL
LIN {X 0,Y 180.488,Z 350.58,A -85,B 0,C 180,E1 -26978.195,E2 -26978.195} C_VEL
LIN {X 0,Y 183.607,Z 336.059,A -85,B 0,C 180,E1 -26978.803,E2 -26978.803} C_VEL
LIN {X 0,Y 185.834,Z 319.368,A -85,B 0,C 180,E1 -26979.268,E2 -26979.268} C_VEL
LIN {X 0,Y 188.674,Z 291.079,A -85,B 0,C 180,E1 -26979.981,E2 -26979.981} C_VEL
LIN {X 0,Y 186.411,Z 285.743,A -85,B 0,C 180,E1 -26982.657,E2 -26982.657} C_VEL
LIN {X 0,Y 184.059,Z 280.619,A -85,B 0,C 180,E1 -26985.977,E2 -26985.977} C_VEL
LIN {X 0,Y 182.418,Z 277.199,A -85,B 0,C 180,E1 -26988.893,E2 -26988.893} C_VEL
LIN {X 0,Y 181.165,Z 274.296,A -85,B 0,C 180,E1 -26991.916,E2 -26991.916} C_VEL
LIN {X 0,Y 179.919,Z 270.536,A -85,B 0,C 180,E1 -26998.321,E2 -26998.321} C_VEL
LIN {X 0,Y 179.895,Z 270.433,A -85,B 0,C 180,E1 -27001.119,E2 -27001.119} C_VEL
LIN {X 0,Y 179.997,Z 271.195,A -85,B 0,C 180,E1 -27002.867,E2 -27002.867} C_VEL
LIN {X 0,Y 181.45,Z 274.925,A -85,B 0,C 180,E1 -27008.772,E2 -27008.772} C_VEL
LIN {X 0,Y 183.11,Z 278.572,A -85,B 0,C 180,E1 -27012.327,E2 -27012.327} C_VEL
LIN {X 0,Y 185.049,Z 282.694,A -85,B 0,C 180,E1 -27015.417,E2 -27015.417} C_VEL
LIN {X 0,Y 187.666,Z 288.533,A -85,B 0,C 180,E1 -27018.774,E2 -27018.774} C_VEL
LIN {X 0,Y 188.712,Z 291.151,A -85,B 0,C 180,E1 -27019.971,E2 -27019.971} C_VEL
LIN {X 0,Y 184.341,Z 332.089,A -85,B 0,C 180,E1 -27020.967,E2 -27020.967} C_VEL
LIN {X 0,Y 181.342,Z 347.838,A -85,B 0,C 180,E1 -27021.544,E2 -27021.544} C_VEL
LIN {X 0,Y 177.119,Z 363.035,A -85,B 0,C 180,E1 -27022.327,E2 -27022.327} C_VEL
LIN {X 0,Y 172.163,Z 376.738,A -85,B 0,C 180,E1 -27023.293,E2 -27023.293} C_VEL
LIN {X 0,Y 166.21,Z 390.161,A -85,B 0,C 180,E1 -27024.618,E2 -27024.618} C_VEL
LIN {X 0,Y 159.43,Z 402.938,A -85,B 0,C 180,E1 -27026.301,E2 -27026.301} C_VEL
LIN {X 0,Y 151.752,Z 415.137,A -85,B 0,C 180,E1 -27028.365,E2 -27028.365} C_VEL
LIN {X 0,Y 143.378,Z 426.583,A -85,B 0,C 180,E1 -27030.929,E2 -27030.929} C_VEL
LIN {X 0,Y 135.346,Z 436.215,A -85,B 0,C 180,E1 -27033.817,E2 -27033.817} C_VEL
LIN {X 0,Y 126.624,Z 445.582,A -85,B 0,C 180,E1 -27037.628,E2 -27037.628} C_VEL
LIN {X 0,Y 118.46,Z 453.561,A -85,B 0,C 180,E1 -27042.132,E2 -27042.132} C_VEL
LIN {X 0,Y 110.005,Z 460.919,A -85,B 0,C 180,E1 -27047.869,E2 -27047.869} C_VEL
LIN {X 0,Y 102.763,Z 466.881,A -85,B 0,C 180,E1 -27054.697,E2 -27054.697} C_VEL
LIN {X 0,Y 98.61,Z 470.23,A -85,B 0,C 180,E1 -27060.073,E2 -27060.073} C_VEL
LIN {X 0,Y 94.196,Z 473.735,A -85,B 0,C 180,E1 -27068.096,E2 -27068.096} C_VEL
LIN {X 0,Y 91.663,Z 476.042,A -85,B 0,C 180,E1 -27076.702,E2 -27076.702} C_VEL
LIN {X 0,Y 90.795,Z 477.201,A -85,B 0,C 180,E1 -27085.56,E2 -27085.56} C_VEL
LIN {X 0,Y 90.839,Z 477.353,A -85,B 0,C 180,E1 -27090,E2 -27090} C_VEL
LIN {X 0,Y 91.06,Z 476.742,A -85,B 0,C 180,E1 -27098.879,E2 -27098.879} C_VEL
LIN {X 0,Y 92.717,Z 474.986,A -85,B 0,C 180,E1 -27107.65,E2 -27107.65} C_VEL
LIN {X 0,Y 96.199,Z 472.065,A -85,B 0,C 180,E1 -27115.998,E2 -27115.998} C_VEL
LIN {X 0,Y 101.359,Z 467.909,A -85,B 0,C 180,E1 -27123.69,E2 -27123.69} C_VEL
LIN {X 0,Y 104.667,Z 465.203,A -85,B 0,C 180,E1 -27127.403,E2 -27127.403} C_VEL
LIN {X 0,Y 106.83,Z 463.046,A -85,B 0,C 180,E1 -27130.132,E2 -27130.132} C_VEL
LIN {X 0,Y 109.359,Z 459.238,A -85,B 0,C 180,E1 -27134.805,E2 -27134.805} C_VEL
LIN {X 0,Y 112.379,Z 455.025,A -85,B 0,C 180,E1 -27139.173,E2 -27139.173} C_VEL
LIN {X 0,Y 115.185,Z 452.105,A -85,B 0,C 180,E1 -27141.341,E2 -27141.341} C_VEL
LIN {X 0,Y 123.518,Z 444.178,A -85,B 0,C 180,E1 -27145.589,E2 -27145.589} C_VEL
LIN {X 0,Y 132.895,Z 434.42,A -85,B 0,C 180,E1 -27149.245,E2 -27149.245} C_VEL
LIN {X 0,Y 141.235,Z 424.44,A -85,B 0,C 180,E1 -27152.038,E2 -27152.038} C_VEL
LIN {X 0,Y 149.96,Z 412.587,A -85,B 0,C 180,E1 -27154.444,E2 -27154.444} C_VEL
LIN {X 0,Y 157.309,Z 400.825,A -85,B 0,C 180,E1 -27156.292,E2 -27156.292} C_VEL
LIN {X 0,Y 164.114,Z 387.985,A -85,B 0,C 180,E1 -27157.83,E2 -27157.83} C_VEL
LIN {X 0,Y 170.236,Z 374.028,A -85,B 0,C 180,E1 -27159.075,E2 -27159.075} C_VEL
LIN {X 0,Y 175.307,Z 359.638,A -85,B 0,C 180,E1 -27159.985,E2 -27159.985} C_VEL
LIN {X 0,Y 179.327,Z 344.414,A -85,B 0,C 180,E1 -27160.674,E2 -27160.674} C_VEL
LIN {X 0,Y 182.067,Z 329.007,A -85,B 0,C 180,E1 -27161.148,E2 -27161.148} C_VEL
LIN {X 0,Y 185.714,Z 294.788,A -85,B 0,C 180,E1 -27161.989,E2 -27161.989} C_VEL
LIN {X 0,Y 183.318,Z 289.001,A -85,B 0,C 180,E1 -27165.287,E2 -27165.287} C_VEL
LIN {X 0,Y 181.303,Z 284.315,A -85,B 0,C 180,E1 -27168.824,E2 -27168.824} C_VEL
LIN {X 0,Y 179.828,Z 280.983,A -85,B 0,C 180,E1 -27172.421,E2 -27172.421} C_VEL
LIN {X 0,Y 178.743,Z 277.427,A -85,B 0,C 180,E1 -27178.31,E2 -27178.31} C_VEL
LIN {X 0,Y 178.697,Z 277.339,A -85,B 0,C 180,E1 -27181.127,E2 -27181.127} C_VEL
LIN {X 0,Y 178.802,Z 277.724,A -85,B 0,C 180,E1 -27182.676,E2 -27182.676} C_VEL
LIN {X 0,Y 179.767,Z 280.892,A -85,B 0,C 180,E1 -27187.582,E2 -27187.582} C_VEL
LIN {X 0,Y 180.349,Z 282.386,A -85,B 0,C 180,E1 -27189.251,E2 -27189.251} C_VEL
LIN {X 0,Y 181.726,Z 285.482,A -85,B 0,C 180,E1 -27192.221,E2 -27192.221} C_VEL
LIN {X 0,Y 183.836,Z 290.227,A -85,B 0,C 180,E1 -27195.664,E2 -27195.664} C_VEL
LIN {X 0,Y 185.712,Z 294.844,A -85,B 0,C 180,E1 -27198.193,E2 -27198.193} C_VEL
LIN {X 0,Y 181.661,Z 331.579,A -85,B 0,C 180,E1 -27199.092,E2 -27199.092} C_VEL
LIN {X 0,Y 178.602,Z 347.018,A -85,B 0,C 180,E1 -27199.619,E2 -27199.619} C_VEL
LIN {X 0,Y 174.344,Z 362.104,A -85,B 0,C 180,E1 -27200.408,E2 -27200.408} C_VEL
LIN {X 0,Y 168.964,Z 376.618,A -85,B 0,C 180,E1 -27201.458,E2 -27201.458} C_VEL
LIN {X 0,Y 162.751,Z 390.152,A -85,B 0,C 180,E1 -27202.791,E2 -27202.791} C_VEL
LIN {X 0,Y 155.49,Z 403.319,A -85,B 0,C 180,E1 -27204.546,E2 -27204.546} C_VEL
LIN {X 0,Y 147.391,Z 415.546,A -85,B 0,C 180,E1 -27206.613,E2 -27206.613} C_VEL
LIN {X 0,Y 138.867,Z 426.689,A -85,B 0,C 180,E1 -27209.189,E2 -27209.189} C_VEL
LIN {X 0,Y 129.263,Z 437.509,A -85,B 0,C 180,E1 -27212.57,E2 -27212.57} C_VEL
LIN {X 0,Y 121.595,Z 445.277,A -85,B 0,C 180,E1 -27215.984,E2 -27215.984} C_VEL
LIN {X 0,Y 113.062,Z 452.94,A -85,B 0,C 180,E1 -27220.406,E2 -27220.406} C_VEL
LIN {X 0,Y 105.362,Z 459.296,A -85,B 0,C 180,E1 -27225.542,E2 -27225.542} C_VEL
LIN {X 0,Y 97.347,Z 465.34,A -85,B 0,C 180,E1 -27232.576,E2 -27232.576} C_VEL
LIN {X 0,Y 92.922,Z 468.593,A -85,B 0,C 180,E1 -27238.033,E2 -27238.033} C_VEL
LIN {X 0,Y 87.992,Z 472.09,A -85,B 0,C 180,E1 -27246.462,E2 -27246.462} C_VEL
LIN {X 0,Y 85.008,Z 474.396,A -85,B 0,C 180,E1 -27255.64,E2 -27255.64} C_VEL
LIN {X 0,Y 83.8,Z 475.566,A -85,B 0,C 180,E1 -27265.189,E2 -27265.189} C_VEL
LIN {X 0,Y 83.813,Z 475.72,A -85,B 0,C 180,E1 -27270,E2 -27270} C_VEL
LIN {X 0,Y 84.193,Z 475.151,A -85,B 0,C 180,E1 -27279.611,E2 -27279.611} C_VEL
LIN {X 0,Y 86.232,Z 473.458,A -85,B 0,C 180,E1 -27289.027,E2 -27289.027} C_VEL
LIN {X 0,Y 90.241,Z 470.6,A -85,B 0,C 180,E1 -27297.858,E2 -27297.858} C_VEL
LIN {X 0,Y 96.005,Z 466.51,A -85,B 0,C 180,E1 -27305.848,E2 -27305.848} C_VEL
LIN {X 0,Y 103.276,Z 461.088,A -85,B 0,C 180,E1 -27312.884,E2 -27312.884} C_VEL
LIN {X 0,Y 111.831,Z 454.181,A -85,B 0,C 180,E1 -27318.95,E2 -27318.95} C_VEL
LIN {X 0,Y 120.289,Z 446.76,A -85,B 0,C 180,E1 -27323.453,E2 -27323.453} C_VEL
LIN {X 0,Y 129.198,Z 437.815,A -85,B 0,C 180,E1 -27327.476,E2 -27327.476} C_VEL
LIN {X 0,Y 138.788,Z 427.066,A -85,B 0,C 180,E1 -27330.87,E2 -27330.87} C_VEL
LIN {X 0,Y 148.048,Z 414.982,A -85,B 0,C 180,E1 -27333.64,E2 -27333.64} C_VEL
LIN {X 0,Y 156.512,Z 401.993,A -85,B 0,C 180,E1 -27335.806,E2 -27335.806} C_VEL
LIN {X 0,Y 163.605,Z 389.027,A -85,B 0,C 180,E1 -27337.453,E2 -27337.453} C_VEL
LIN {X 0,Y 169.644,Z 375.636,A -85,B 0,C 180,E1 -27338.77,E2 -27338.77} C_VEL
LIN {X 0,Y 175.056,Z 360.806,A -85,B 0,C 180,E1 -27339.791,E2 -27339.791} C_VEL
LIN {X 0,Y 179.319,Z 345.138,A -85,B 0,C 180,E1 -27340.583,E2 -27340.583} C_VEL
LIN {X 0,Y 182.164,Z 330.224,A -85,B 0,C 180,E1 -27341.061,E2 -27341.061} C_VEL
LIN {X 0,Y 185.928,Z 294.95,A -85,B 0,C 180,E1 -27341.977,E2 -27341.977} C_VEL
LIN {X 0,Y 183.717,Z 289.601,A -85,B 0,C 180,E1 -27345.014,E2 -27345.014} C_VEL
LIN {X 0,Y 181.54,Z 284.487,A -85,B 0,C 180,E1 -27348.839,E2 -27348.839} C_VEL
LIN {X 0,Y 180.092,Z 281.165,A -85,B 0,C 180,E1 -27352.431,E2 -27352.431} C_VEL
LIN {X 0,Y 179.05,Z 277.618,A -85,B 0,C 180,E1 -27358.313,E2 -27358.313} C_VEL
LIN {X 0,Y 179.029,Z 277.489,A -85,B 0,C 180,E1 -27361.124,E2 -27361.124} C_VEL
LIN {X 0,Y 179.113,Z 278.405,A -85,B 0,C 180,E1 -27362.881,E2 -27362.881} C_VEL
LIN {X 0,Y 180.358,Z 281.765,A -85,B 0,C 180,E1 -27368.261,E2 -27368.261} C_VEL
LIN {X 0,Y 181.933,Z 285.486,A -85,B 0,C 180,E1 -27371.877,E2 -27371.877} C_VEL
LIN {X 0,Y 183.948,Z 290.029,A -85,B 0,C 180,E1 -27375.228,E2 -27375.228} C_VEL
LIN {X 0,Y 185.976,Z 295.044,A -85,B 0,C 180,E1 -27377.994,E2 -27377.994} C_VEL
LIN {X 0,Y 181.927,Z 332.037,A -85,B 0,C 180,E1 -27378.884,E2 -27378.884} C_VEL
LIN {X 0,Y 178.858,Z 347.781,A -85,B 0,C 180,E1 -27379.429,E2 -27379.429} C_VEL
LIN {X 0,Y 174.543,Z 362.976,A -85,B 0,C 180,E1 -27380.168,E2 -27380.168} C_VEL
LIN {X 0,Y 169.486,Z 376.677,A -85,B 0,C 180,E1 -27381.092,E2 -27381.092} C_VEL
LIN {X 0,Y 163.369,Z 390.099,A -85,B 0,C 180,E1 -27382.344,E2 -27382.344} C_VEL
LIN {X 0,Y 155.942,Z 403.68,A -85,B 0,C 180,E1 -27384.074,E2 -27384.074} C_VEL
LIN {X 0,Y 147.775,Z 416.144,A -85,B 0,C 180,E1 -27386.146,E2 -27386.146} C_VEL
LIN {X 0,Y 139.834,Z 426.519,A -85,B 0,C 180,E1 -27388.413,E2 -27388.413} C_VEL
LIN {X 0,Y 131.504,Z 436.15,A -85,B 0,C 180,E1 -27391.23,E2 -27391.23} C_VEL
LIN {X 0,Y 121.848,Z 446.042,A -85,B 0,C 180,E1 -27395.224,E2 -27395.224} C_VEL
LIN {X 0,Y 112.618,Z 454.506,A -85,B 0,C 180,E1 -27400.14,E2 -27400.14} C_VEL
LIN {X 0,Y 104.806,Z 460.853,A -85,B 0,C 180,E1 -27405.243,E2 -27405.243} C_VEL
LIN {X 0,Y 97.176,Z 466.691,A -85,B 0,C 180,E1 -27412.067,E2 -27412.067} C_VEL
LIN {X 0,Y 92.478,Z 470.164,A -85,B 0,C 180,E1 -27417.86,E2 -27417.86} C_VEL
LIN {X 0,Y 87.609,Z 473.669,A -85,B 0,C 180,E1 -27426.353,E2 -27426.353} C_VEL
LIN {X 0,Y 84.735,Z 475.975,A -85,B 0,C 180,E1 -27435.592,E2 -27435.592} C_VEL
LIN {X 0,Y 83.709,Z 477.134,A -85,B 0,C 180,E1 -27445.184,E2 -27445.184} C_VEL
LIN {X 0,Y 83.76,Z 477.287,A -85,B 0,C 180,E1 -27450,E2 -27450} C_VEL
LIN {X 0,Y 84.023,Z 476.675,A -85,B 0,C 180,E1 -27459.63,E2 -27459.63} C_VEL
LIN {X 0,Y 85.915,Z 474.919,A -85,B 0,C 180,E1 -27469.099,E2 -27469.099} C_VEL
LIN {X 0,Y 89.82,Z 471.997,A -85,B 0,C 180,E1 -27478,E2 -27478} C_VEL
LIN {X 0,Y 95.472,Z 467.841,A -85,B 0,C 180,E1 -27486.079,E2 -27486.079} C_VEL
LIN {X 0,Y 102.747,Z 462.34,A -85,B 0,C 180,E1 -27493.158,E2 -27493.158} C_VEL
LIN {X 0,Y 111.44,Z 455.346,A -85,B 0,C 180,E1 -27499.181,E2 -27499.181} C_VEL
LIN {X 0,Y 115.185,Z 452.105,A -85,B 0,C 180,E1 -27501.341,E2 -27501.341} C_VEL
LIN {X 0,Y 118.059,Z 449.081,A -85,B 0,C 180,E1 -27503.38,E2 -27503.38} C_VEL
LIN {X 0,Y 124.873,Z 439.609,A -85,B 0,C 180,E1 -27509.747,E2 -27509.747} C_VEL
LIN {X 0,Y 127.832,Z 436.024,A -85,B 0,C 180,E1 -27511.403,E2 -27511.403} C_VEL
LIN {X 0,Y 128.993,Z 434.757,A -85,B 0,C 180,E1 -27511.841,E2 -27511.841} C_VEL
LIN {X 0,Y 138.027,Z 424.371,A -85,B 0,C 180,E1 -27514.66,E2 -27514.66} C_VEL
LIN {X 0,Y 147.038,Z 412.517,A -85,B 0,C 180,E1 -27516.94,E2 -27516.94} C_VEL
LIN {X 0,Y 155.162,Z 399.794,A -85,B 0,C 180,E1 -27518.824,E2 -27518.824} C_VEL
LIN {X 0,Y 162.346,Z 386.33,A -85,B 0,C 180,E1 -27520.316,E2 -27520.316} C_VEL
LIN {X 0,Y 168.617,Z 371.969,A -85,B 0,C 180,E1 -27521.482,E2 -27521.482} C_VEL
LIN {X 0,Y 173.412,Z 358.264,A -85,B 0,C 180,E1 -27522.252,E2 -27522.252} C_VEL
LIN {X 0,Y 177.38,Z 343.116,A -85,B 0,C 180,E1 -27522.874,E2 -27522.874} C_VEL
LIN {X 0,Y 180.114,Z 327.174,A -85,B 0,C 180,E1 -27523.343,E2 -27523.343} C_VEL
LIN {X 0,Y 183.206,Z 298.933,A -85,B 0,C 180,E1 -27523.983,E2 -27523.983} C_VEL
LIN {X 0,Y 181.026,Z 293.407,A -85,B 0,C 180,E1 -27527.529,E2 -27527.529} C_VEL
LIN {X 0,Y 179.823,Z 290.511,A -85,B 0,C 180,E1 -27530.013,E2 -27530.013} C_VEL
LIN {X 0,Y 178.815,Z 287.889,A -85,B 0,C 180,E1 -27532.803,E2 -27532.803} C_VEL
LIN {X 0,Y 177.875,Z 284.496,A -85,B 0,C 180,E1 -27538.302,E2 -27538.302} C_VEL
LIN {X 0,Y 177.832,Z 284.385,A -85,B 0,C 180,E1 -27541.133,E2 -27541.133} C_VEL
LIN {X 0,Y 177.903,Z 284.897,A -85,B 0,C 180,E1 -27542.547,E2 -27542.547} C_VEL
LIN {X 0,Y 179.064,Z 288.624,A -85,B 0,C 180,E1 -27548.18,E2 -27548.18} C_VEL
LIN {X 0,Y 180.463,Z 292.219,A -85,B 0,C 180,E1 -27551.588,E2 -27551.588} C_VEL
LIN {X 0,Y 182.257,Z 296.541,A -85,B 0,C 180,E1 -27554.766,E2 -27554.766} C_VEL
LIN {X 0,Y 183.172,Z 298.895,A -85,B 0,C 180,E1 -27556.151,E2 -27556.151} C_VEL
LIN {X 0,Y 179.463,Z 331.66,A -85,B 0,C 180,E1 -27556.948,E2 -27556.948} C_VEL
LIN {X 0,Y 176.342,Z 347.094,A -85,B 0,C 180,E1 -27557.444,E2 -27557.444} C_VEL
LIN {X 0,Y 172.003,Z 362.177,A -85,B 0,C 180,E1 -27558.197,E2 -27558.197} C_VEL
LIN {X 0,Y 166.494,Z 376.691,A -85,B 0,C 180,E1 -27559.181,E2 -27559.181} C_VEL
LIN {X 0,Y 159.937,Z 390.575,A -85,B 0,C 180,E1 -27560.48,E2 -27560.48} C_VEL
LIN {X 0,Y 152.636,Z 403.443,A -85,B 0,C 180,E1 -27562.124,E2 -27562.124} C_VEL
LIN {X 0,Y 144.336,Z 415.615,A -85,B 0,C 180,E1 -27564.081,E2 -27564.081} C_VEL
LIN {X 0,Y 135.526,Z 426.758,A -85,B 0,C 180,E1 -27566.551,E2 -27566.551} C_VEL
LIN {X 0,Y 125.565,Z 437.578,A -85,B 0,C 180,E1 -27569.825,E2 -27569.825} C_VEL
LIN {X 0,Y 116.241,Z 446.564,A -85,B 0,C 180,E1 -27573.764,E2 -27573.764} C_VEL
LIN {X 0,Y 107.331,Z 454.013,A -85,B 0,C 180,E1 -27578.209,E2 -27578.209} C_VEL
LIN {X 0,Y 98.203,Z 460.973,A -85,B 0,C 180,E1 -27584.303,E2 -27584.303} C_VEL
LIN {X 0,Y 90.273,Z 466.44,A -85,B 0,C 180,E1 -27591.478,E2 -27591.478} C_VEL
LIN {X 0,Y 84.01,Z 470.562,A -85,B 0,C 180,E1 -27599.872,E2 -27599.872} C_VEL
LIN {X 0,Y 79.569,Z 473.454,A -85,B 0,C 180,E1 -27609.311,E2 -27609.311} C_VEL
LIN {X 0,Y 77.202,Z 475.187,A -85,B 0,C 180,E1 -27619.51,E2 -27619.51} C_VEL
LIN {X 0,Y 76.734,Z 475.787,A -85,B 0,C 180,E1 -27630,E2 -27630} C_VEL
LIN {X 0,Y 77.196,Z 475.217,A -85,B 0,C 180,E1 -27640.491,E2 -27640.491} C_VEL
LIN {X 0,Y 79.529,Z 473.524,A -85,B 0,C 180,E1 -27650.701,E2 -27650.701} C_VEL
LIN {X 0,Y 83.985,Z 470.666,A -85,B 0,C 180,E1 -27660.139,E2 -27660.139} C_VEL
LIN {X 0,Y 90.293,Z 466.576,A -85,B 0,C 180,E1 -27668.513,E2 -27668.513} C_VEL
LIN {X 0,Y 98.152,Z 461.154,A -85,B 0,C 180,E1 -27675.728,E2 -27675.728} C_VEL
LIN {X 0,Y 107.273,Z 454.246,A -85,B 0,C 180,E1 -27681.83,E2 -27681.83} C_VEL
LIN {X 0,Y 116.17,Z 446.825,A -85,B 0,C 180,E1 -27686.289,E2 -27686.289} C_VEL
LIN {X 0,Y 125.504,Z 437.879,A -85,B 0,C 180,E1 -27690.224,E2 -27690.224} C_VEL
LIN {X 0,Y 135.452,Z 427.13,A -85,B 0,C 180,E1 -27693.512,E2 -27693.512} C_VEL
LIN {X 0,Y 145.033,Z 415.045,A -85,B 0,C 180,E1 -27696.156,E2 -27696.156} C_VEL
LIN {X 0,Y 153.003,Z 403.255,A -85,B 0,C 180,E1 -27698.06,E2 -27698.06} C_VEL
LIN {X 0,Y 160.238,Z 390.562,A -85,B 0,C 180,E1 -27699.637,E2 -27699.637} C_VEL
LIN {X 0,Y 166.42,Z 377.474,A -85,B 0,C 180,E1 -27700.893,E2 -27700.893} C_VEL
LIN {X 0,Y 171.562,Z 364.286,A -85,B 0,C 180,E1 -27701.782,E2 -27701.782} C_VEL
LIN {X 0,Y 176.097,Z 349.17,A -85,B 0,C 180,E1 -27702.572,E2 -27702.572} C_VEL
LIN {X 0,Y 179.225,Z 334.712,A -85,B 0,C 180,E1 -27703.077,E2 -27703.077} C_VEL
LIN {X 0,Y 181.823,Z 314.527,A -85,B 0,C 180,E1 -27703.578,E2 -27703.578} C_VEL
LIN {X 0,Y 183.445,Z 299.104,A -85,B 0,C 180,E1 -27703.956,E2 -27703.956} C_VEL
LIN {X 0,Y 181.381,Z 293.903,A -85,B 0,C 180,E1 -27707.304,E2 -27707.304} C_VEL
LIN {X 0,Y 179.946,Z 290.473,A -85,B 0,C 180,E1 -27710.303,E2 -27710.303} C_VEL
LIN {X 0,Y 178.95,Z 287.848,A -85,B 0,C 180,E1 -27713.233,E2 -27713.233} C_VEL
LIN {X 0,Y 178.155,Z 284.564,A -85,B 0,C 180,E1 -27718.87,E2 -27718.87} C_VEL
LIN {X 0,Y 178.176,Z 284.601,A -85,B 0,C 180,E1 -27721.412,E2 -27721.412} C_VEL
LIN {X 0,Y 179.28,Z 288.604,A -85,B 0,C 180,E1 -27727.744,E2 -27727.744} C_VEL
LIN {X 0,Y 180.665,Z 292.178,A -85,B 0,C 180,E1 -27731.215,E2 -27731.215} C_VEL
LIN {X 0,Y 182.365,Z 296.272,A -85,B 0,C 180,E1 -27734.293,E2 -27734.293} C_VEL
LIN {X 0,Y 183.464,Z 299.141,A -85,B 0,C 180,E1 -27735.984,E2 -27735.984} C_VEL
LIN {X 0,Y 179.855,Z 331.384,A -85,B 0,C 180,E1 -27736.732,E2 -27736.732} C_VEL
LIN {X 0,Y 176.85,Z 346.835,A -85,B 0,C 180,E1 -27737.226,E2 -27737.226} C_VEL
LIN {X 0,Y 172.624,Z 361.739,A -85,B 0,C 180,E1 -27737.887,E2 -27737.887} C_VEL
LIN {X 0,Y 167.065,Z 376.617,A -85,B 0,C 180,E1 -27738.823,E2 -27738.823} C_VEL
LIN {X 0,Y 160.796,Z 390.038,A -85,B 0,C 180,E1 -27739.996,E2 -27739.996} C_VEL
LIN {X 0,Y 153.155,Z 403.617,A -85,B 0,C 180,E1 -27741.623,E2 -27741.623} C_VEL
LIN {X 0,Y 144.78,Z 416.08,A -85,B 0,C 180,E1 -27743.616,E2 -27743.616} C_VEL
LIN {X 0,Y 136.586,Z 426.455,A -85,B 0,C 180,E1 -27745.781,E2 -27745.781} C_VEL
LIN {X 0,Y 127.953,Z 436.086,A -85,B 0,C 180,E1 -27748.498,E2 -27748.498} C_VEL
LIN {X 0,Y 119.406,Z 444.56,A -85,B 0,C 180,E1 -27751.733,E2 -27751.733} C_VEL
LIN {X 0,Y 110.628,Z 452.42,A -85,B 0,C 180,E1 -27755.905,E2 -27755.905} C_VEL
LIN {X 0,Y 102.095,Z 459.124,A -85,B 0,C 180,E1 -27760.78,E2 -27760.78} C_VEL
LIN {X 0,Y 93.531,Z 465.312,A -85,B 0,C 180,E1 -27767.447,E2 -27767.447} C_VEL
LIN {X 0,Y 86.501,Z 470.098,A -85,B 0,C 180,E1 -27775.338,E2 -27775.338} C_VEL
LIN {X 0,Y 81.121,Z 473.603,A -85,B 0,C 180,E1 -27784.33,E2 -27784.33} C_VEL
LIN {X 0,Y 77.85,Z 475.909,A -85,B 0,C 180,E1 -27794.286,E2 -27794.286} C_VEL
LIN {X 0,Y 76.614,Z 477.068,A -85,B 0,C 180,E1 -27804.736,E2 -27804.736} C_VEL
LIN {X 0,Y 76.671,Z 477.221,A -85,B 0,C 180,E1 -27810,E2 -27810} C_VEL
LIN {X 0,Y 76.993,Z 476.608,A -85,B 0,C 180,E1 -27820.519,E2 -27820.519} C_VEL
LIN {X 0,Y 79.181,Z 474.851,A -85,B 0,C 180,E1 -27830.795,E2 -27830.795} C_VEL
LIN {X 0,Y 83.557,Z 471.93,A -85,B 0,C 180,E1 -27840.309,E2 -27840.309} C_VEL
LIN {X 0,Y 89.764,Z 467.773,A -85,B 0,C 180,E1 -27848.782,E2 -27848.782} C_VEL
LIN {X 0,Y 97.658,Z 462.272,A -85,B 0,C 180,E1 -27856.026,E2 -27856.026} C_VEL
LIN {X 0,Y 106.906,Z 455.277,A -85,B 0,C 180,E1 -27862.081,E2 -27862.081} C_VEL
LIN {X 0,Y 115.398,Z 447.992,A -85,B 0,C 180,E1 -27866.593,E2 -27866.593} C_VEL
LIN {X 0,Y 125.14,Z 438.775,A -85,B 0,C 180,E1 -27870.517,E2 -27870.517} C_VEL
LIN {X 0,Y 128.993,Z 434.757,A -85,B 0,C 180,E1 -27871.841,E2 -27871.841} C_VEL
LIN {X 0,Y 132.205,Z 430.957,A -85,B 0,C 180,E1 -27873.244,E2 -27873.244} C_VEL
LIN {X 0,Y 136.402,Z 424.615,A -85,B 0,C 180,E1 -27875.972,E2 -27875.972} C_VEL
LIN {X 0,Y 140.591,Z 417.894,A -85,B 0,C 180,E1 -27878.418,E2 -27878.418} C_VEL
LIN {X 0,Y 143.658,Z 413.459,A -85,B 0,C 180,E1 -27879.384,E2 -27879.384} C_VEL
LIN {X 0,Y 151.257,Z 402.154,A -85,B 0,C 180,E1 -27881.02,E2 -27881.02} C_VEL
LIN {X 0,Y 158.499,Z 389.426,A -85,B 0,C 180,E1 -27882.426,E2 -27882.426} C_VEL
LIN {X 0,Y 164.895,Z 375.87,A -85,B 0,C 180,E1 -27883.532,E2 -27883.532} C_VEL
LIN {X 0,Y 170.56,Z 360.789,A -85,B 0,C 180,E1 -27884.403,E2 -27884.403} C_VEL
LIN {X 0,Y 174.773,Z 345.943,A -85,B 0,C 180,E1 -27885.001,E2 -27885.001} C_VEL
LIN {X 0,Y 177.773,Z 330.442,A -85,B 0,C 180,E1 -27885.444,E2 -27885.444} C_VEL
LIN {X 0,Y 180.837,Z 303.952,A -85,B 0,C 180,E1 -27886.003,E2 -27886.003} C_VEL
LIN {X 0,Y 180.879,Z 303.239,A -85,B 0,C 180,E1 -27886.063,E2 -27886.063} C_VEL
LIN {X 0,Y 179.286,Z 298.94,A -85,B 0,C 180,E1 -27889.126,E2 -27889.126} C_VEL
LIN {X 0,Y 177.893,Z 295.006,A -85,B 0,C 180,E1 -27892.908,E2 -27892.908} C_VEL
LIN {X 0,Y 176.978,Z 291.427,A -85,B 0,C 180,E1 -27898.863,E2 -27898.863} C_VEL
LIN {X 0,Y 177.001,Z 291.592,A -85,B 0,C 180,E1 -27901.849,E2 -27901.849} C_VEL
LIN {X 0,Y 177.951,Z 295.336,A -85,B 0,C 180,E1 -27907.517,E2 -27907.517} C_VEL
LIN {X 0,Y 179.136,Z 298.667,A -85,B 0,C 180,E1 -27910.74,E2 -27910.74} C_VEL
LIN {X 0,Y 180.759,Z 302.953,A -85,B 0,C 180,E1 -27913.913,E2 -27913.913} C_VEL
LIN {X 0,Y 180.874,Z 303.281,A -85,B 0,C 180,E1 -27914.114,E2 -27914.114} C_VEL
LIN {X 0,Y 177.436,Z 332.279,A -85,B 0,C 180,E1 -27914.78,E2 -27914.78} C_VEL
LIN {X 0,Y 174.347,Z 347.17,A -85,B 0,C 180,E1 -27915.218,E2 -27915.218} C_VEL
LIN {X 0,Y 169.924,Z 362.251,A -85,B 0,C 180,E1 -27915.927,E2 -27915.927} C_VEL
LIN {X 0,Y 164.293,Z 376.763,A -85,B 0,C 180,E1 -27916.835,E2 -27916.835} C_VEL
LIN {X 0,Y 157.861,Z 390.15,A -85,B 0,C 180,E1 -27918.002,E2 -27918.002} C_VEL
LIN {X 0,Y 150.055,Z 403.578,A -85,B 0,C 180,E1 -27919.613,E2 -27919.613} C_VEL
LIN {X 0,Y 141.585,Z 415.685,A -85,B 0,C 180,E1 -27921.453,E2 -27921.453} C_VEL
LIN {X 0,Y 132.485,Z 426.828,A -85,B 0,C 180,E1 -27923.785,E2 -27923.785} C_VEL
LIN {X 0,Y 122.182,Z 437.647,A -85,B 0,C 180,E1 -27926.929,E2 -27926.929} C_VEL
LIN {X 0,Y 113.755,Z 445.415,A -85,B 0,C 180,E1 -27930.123,E2 -27930.123} C_VEL
LIN {X 0,Y 104.367,Z 453.077,A -85,B 0,C 180,E1 -27934.421,E2 -27934.421} C_VEL
LIN {X 0,Y 95.689,Z 459.432,A -85,B 0,C 180,E1 -27939.54,E2 -27939.54} C_VEL
LIN {X 0,Y 86.774,Z 465.273,A -85,B 0,C 180,E1 -27946.497,E2 -27946.497} C_VEL
LIN {X 0,Y 81.133,Z 468.728,A -85,B 0,C 180,E1 -27952.673,E2 -27952.673} C_VEL
LIN {X 0,Y 75.104,Z 472.225,A -85,B 0,C 180,E1 -27962.103,E2 -27962.103} C_VEL
LIN {X 0,Y 71.286,Z 474.53,A -85,B 0,C 180,E1 -27972.797,E2 -27972.797} C_VEL
LIN {X 0,Y 69.655,Z 475.699,A -85,B 0,C 180,E1 -27984.209,E2 -27984.209} C_VEL
LIN {X 0,Y 69.646,Z 475.853,A -85,B 0,C 180,E1 -27990,E2 -27990} C_VEL
LIN {X 0,Y 70.205,Z 475.283,A -85,B 0,C 180,E1 -28001.55,E2 -28001.55} C_VEL
LIN {X 0,Y 72.893,Z 473.59,A -85,B 0,C 180,E1 -28012.685,E2 -28012.685} C_VEL
LIN {X 0,Y 77.889,Z 470.732,A -85,B 0,C 180,E1 -28022.778,E2 -28022.778} C_VEL
LIN {X 0,Y 85.555,Z 466.155,A -85,B 0,C 180,E1 -28032.326,E2 -28032.326} C_VEL
LIN {X 0,Y 93.308,Z 461.219,A -85,B 0,C 180,E1 -28038.869,E2 -28038.869} C_VEL
LIN {X 0,Y 103.015,Z 454.311,A -85,B 0,C 180,E1 -28044.953,E2 -28044.953} C_VEL
LIN {X 0,Y 112.345,Z 446.89,A -85,B 0,C 180,E1 -28049.336,E2 -28049.336} C_VEL
LIN {X 0,Y 122.124,Z 437.943,A -85,B 0,C 180,E1 -28053.126,E2 -28053.126} C_VEL
LIN {X 0,Y 132.427,Z 427.194,A -85,B 0,C 180,E1 -28056.274,E2 -28056.274} C_VEL
LIN {X 0,Y 142.305,Z 415.108,A -85,B 0,C 180,E1 -28058.778,E2 -28058.778} C_VEL
LIN {X 0,Y 150.374,Z 403.494,A -85,B 0,C 180,E1 -28060.546,E2 -28060.546} C_VEL
LIN {X 0,Y 157.906,Z 390.623,A -85,B 0,C 180,E1 -28062.055,E2 -28062.055} C_VEL
LIN {X 0,Y 164.232,Z 377.535,A -85,B 0,C 180,E1 -28063.236,E2 -28063.236} C_VEL
LIN {X 0,Y 169.477,Z 364.346,A -85,B 0,C 180,E1 -28064.062,E2 -28064.062} C_VEL
LIN {X 0,Y 174.103,Z 349.227,A -85,B 0,C 180,E1 -28064.802,E2 -28064.802} C_VEL
LIN {X 0,Y 177.404,Z 334.124,A -85,B 0,C 180,E1 -28065.287,E2 -28065.287} C_VEL
LIN {X 0,Y 180.087,Z 313.219,A -85,B 0,C 180,E1 -28065.783,E2 -28065.783} C_VEL
LIN {X 0,Y 181.132,Z 303.461,A -85,B 0,C 180,E1 -28066.024,E2 -28066.024} C_VEL
LIN {X 0,Y 179.646,Z 299.504,A -85,B 0,C 180,E1 -28068.862,E2 -28068.862} C_VEL
LIN {X 0,Y 178.624,Z 296.783,A -85,B 0,C 180,E1 -28071.373,E2 -28071.373} C_VEL
LIN {X 0,Y 177.927,Z 294.739,A -85,B 0,C 180,E1 -28073.718,E2 -28073.718} C_VEL
LIN {X 0,Y 177.288,Z 291.626,A -85,B 0,C 180,E1 -28078.864,E2 -28078.864} C_VEL
LIN {X 0,Y 177.294,Z 291.696,A -85,B 0,C 180,E1 -28081.277,E2 -28081.277} C_VEL
LIN {X 0,Y 178.245,Z 295.566,A -85,B 0,C 180,E1 -28087.327,E2 -28087.327} C_VEL
LIN {X 0,Y 179.409,Z 298.806,A -85,B 0,C 180,E1 -28090.51,E2 -28090.51} C_VEL
LIN {X 0,Y 180.939,Z 302.852,A -85,B 0,C 180,E1 -28093.541,E2 -28093.541} C_VEL
LIN {X 0,Y 181.151,Z 303.48,A -85,B 0,C 180,E1 -28093.917,E2 -28093.917} C_VEL
LIN {X 0,Y 177.815,Z 332.088,A -85,B 0,C 180,E1 -28094.557,E2 -28094.557} C_VEL
LIN {X 0,Y 174.65,Z 347.667,A -85,B 0,C 180,E1 -28095.033,E2 -28095.033} C_VEL
LIN {X 0,Y 170.176,Z 362.858,A -85,B 0,C 180,E1 -28095.683,E2 -28095.683} C_VEL
LIN {X 0,Y 164.915,Z 376.557,A -85,B 0,C 180,E1 -28096.492,E2 -28096.492} C_VEL
LIN {X 0,Y 158.5,Z 389.976,A -85,B 0,C 180,E1 -28097.574,E2 -28097.574} C_VEL
LIN {X 0,Y 151.224,Z 402.643,A -85,B 0,C 180,E1 -28098.985,E2 -28098.985} C_VEL
LIN {X 0,Y 142.846,Z 414.948,A -85,B 0,C 180,E1 -28100.803,E2 -28100.803} C_VEL
LIN {X 0,Y 133.639,Z 426.391,A -85,B 0,C 180,E1 -28103.027,E2 -28103.027} C_VEL
LIN {X 0,Y 124.706,Z 436.022,A -85,B 0,C 180,E1 -28105.616,E2 -28105.616} C_VEL
LIN {X 0,Y 114.683,Z 445.483,A -85,B 0,C 180,E1 -28109.159,E2 -28109.159} C_VEL
LIN {X 0,Y 105.273,Z 453.365,A -85,B 0,C 180,E1 -28113.436,E2 -28113.436} C_VEL
LIN {X 0,Y 95.166,Z 460.722,A -85,B 0,C 180,E1 -28119.156,E2 -28119.156} C_VEL
LIN {X 0,Y 86.325,Z 466.559,A -85,B 0,C 180,E1 -28126.21,E2 -28126.21} C_VEL
LIN {X 0,Y 80.702,Z 470.032,A -85,B 0,C 180,E1 -28132.439,E2 -28132.439} C_VEL
LIN {X 0,Y 74.752,Z 473.537,A -85,B 0,C 180,E1 -28141.96,E2 -28141.96} C_VEL
LIN {X 0,Y 70.987,Z 475.843,A -85,B 0,C 180,E1 -28152.721,E2 -28152.721} C_VEL
LIN {X 0,Y 69.538,Z 477.001,A -85,B 0,C 180,E1 -28164.199,E2 -28164.199} C_VEL
LIN {X 0,Y 69.571,Z 477.154,A -85,B 0,C 180,E1 -28170,E2 -28170} C_VEL
LIN {X 0,Y 69.999,Z 476.541,A -85,B 0,C 180,E1 -28181.584,E2 -28181.584} C_VEL
LIN {X 0,Y 72.532,Z 474.784,A -85,B 0,C 180,E1 -28192.804,E2 -28192.804} C_VEL
LIN {X 0,Y 77.453,Z 471.862,A -85,B 0,C 180,E1 -28202.986,E2 -28202.986} C_VEL
LIN {X 0,Y 84.303,Z 467.705,A -85,B 0,C 180,E1 -28211.83,E2 -28211.83} C_VEL
LIN {X 0,Y 92.818,Z 462.204,A -85,B 0,C 180,E1 -28219.216,E2 -28219.216} C_VEL
LIN {X 0,Y 102.658,Z 455.209,A -85,B 0,C 180,E1 -28225.237,E2 -28225.237} C_VEL
LIN {X 0,Y 112.101,Z 447.49,A -85,B 0,C 180,E1 -28229.898,E2 -28229.898} C_VEL
LIN {X 0,Y 121.779,Z 438.706,A -85,B 0,C 180,E1 -28233.447,E2 -28233.447} C_VEL
LIN {X 0,Y 132.118,Z 427.858,A -85,B 0,C 180,E1 -28236.579,E2 -28236.579} C_VEL
LIN {X 0,Y 141.282,Z 416.69,A -85,B 0,C 180,E1 -28238.861,E2 -28238.861} C_VEL
LIN {X 0,Y 143.658,Z 413.459,A -85,B 0,C 180,E1 -28239.384,E2 -28239.384} C_VEL
LIN {X 0,Y 146.669,Z 408.956,A -85,B 0,C 180,E1 -28240.293,E2 -28240.293} C_VEL
LIN {X 0,Y 150.618,Z 401.534,A -85,B 0,C 180,E1 -28242.339,E2 -28242.339} C_VEL
LIN {X 0,Y 154.295,Z 393.828,A -85,B 0,C 180,E1 -28244.247,E2 -28244.247} C_VEL
LIN {X 0,Y 156.775,Z 388.817,A -85,B 0,C 180,E1 -28244.953,E2 -28244.953} C_VEL
LIN {X 0,Y 163.023,Z 375.797,A -85,B 0,C 180,E1 -28245.927,E2 -28245.927} C_VEL
LIN {X 0,Y 168.792,Z 360.714,A -85,B 0,C 180,E1 -28246.722,E2 -28246.722} C_VEL
LIN {X 0,Y 173.138,Z 345.574,A -85,B 0,C 180,E1 -28247.28,E2 -28247.28} C_VEL
LIN {X 0,Y 176.165,Z 330.052,A -85,B 0,C 180,E1 -28247.684,E2 -28247.684} C_VEL
LIN {X 0,Y 178.801,Z 307.777,A -85,B 0,C 180,E1 -28248.144,E2 -28248.144} C_VEL
LIN {X 0,Y 177.481,Z 303.907,A -85,B 0,C 180,E1 -28251.317,E2 -28251.317} C_VEL
LIN {X 0,Y 176.699,Z 301.521,A -85,B 0,C 180,E1 -28253.987,E2 -28253.987} C_VEL
LIN {X 0,Y 176.108,Z 298.514,A -85,B 0,C 180,E1 -28258.857,E2 -28258.857} C_VEL
LIN {X 0,Y 176.101,Z 298.485,A -85,B 0,C 180,E1 -28261.144,E2 -28261.144} C_VEL
LIN {X 0,Y 176.897,Z 302.195,A -85,B 0,C 180,E1 -28266.989,E2 -28266.989} C_VEL
LIN {X 0,Y 178.045,Z 305.714,A -85,B 0,C 180,E1 -28270.376,E2 -28270.376} C_VEL
LIN {X 0,Y 178.775,Z 307.802,A -85,B 0,C 180,E1 -28271.998,E2 -28271.998} C_VEL
LIN {X 0,Y 175.757,Z 332.362,A -85,B 0,C 180,E1 -28272.539,E2 -28272.539} C_VEL
LIN {X 0,Y 172.622,Z 347.246,A -85,B 0,C 180,E1 -28272.948,E2 -28272.948} C_VEL
LIN {X 0,Y 168.119,Z 362.324,A -85,B 0,C 180,E1 -28273.606,E2 -28273.606} C_VEL
LIN {X 0,Y 162.375,Z 376.835,A -85,B 0,C 180,E1 -28274.432,E2 -28274.432} C_VEL
LIN {X 0,Y 155.898,Z 390.073,A -85,B 0,C 180,E1 -28275.506,E2 -28275.506} C_VEL
LIN {X 0,Y 148.429,Z 402.737,A -85,B 0,C 180,E1 -28276.909,E2 -28276.909} C_VEL
LIN {X 0,Y 139.144,Z 415.755,A -85,B 0,C 180,E1 -28278.73,E2 -28278.73} C_VEL
LIN {X 0,Y 129.775,Z 426.897,A -85,B 0,C 180,E1 -28280.904,E2 -28280.904} C_VEL
LIN {X 0,Y 119.114,Z 437.716,A -85,B 0,C 180,E1 -28283.861,E2 -28283.861} C_VEL
LIN {X 0,Y 108.929,Z 446.702,A -85,B 0,C 180,E1 -28287.485,E2 -28287.485} C_VEL
LIN {X 0,Y 99.129,Z 454.15,A -85,B 0,C 180,E1 -28291.704,E2 -28291.704} C_VEL
LIN {X 0,Y 88.819,Z 461.109,A -85,B 0,C 180,E1 -28297.696,E2 -28297.696} C_VEL
LIN {X 0,Y 79.547,Z 466.576,A -85,B 0,C 180,E1 -28305.025,E2 -28305.025} C_VEL
LIN {X 0,Y 72.008,Z 470.697,A -85,B 0,C 180,E1 -28314.155,E2 -28314.155} C_VEL
LIN {X 0,Y 66.4,Z 473.589,A -85,B 0,C 180,E1 -28324.953,E2 -28324.953} C_VEL
LIN {X 0,Y 63.239,Z 475.321,A -85,B 0,C 180,E1 -28337.158,E2 -28337.158} C_VEL
LIN {X 0,Y 62.547,Z 475.919,A -85,B 0,C 180,E1 -28350,E2 -28350} C_VEL
LIN {X 0,Y 63.232,Z 475.35,A -85,B 0,C 180,E1 -28362.844,E2 -28362.844} C_VEL
LIN {X 0,Y 66.349,Z 473.657,A -85,B 0,C 180,E1 -28375.069,E2 -28375.069} C_VEL
LIN {X 0,Y 71.991,Z 470.798,A -85,B 0,C 180,E1 -28385.856,E2 -28385.856} C_VEL
LIN {X 0,Y 79.879,Z 466.526,A -85,B 0,C 180,E1 -28395.261,E2 -28395.261} C_VEL
LIN {X 0,Y 88.757,Z 461.285,A -85,B 0,C 180,E1 -28402.357,E2 -28402.357} C_VEL
LIN {X 0,Y 99.087,Z 454.377,A -85,B 0,C 180,E1 -28408.335,E2 -28408.335} C_VEL
LIN {X 0,Y 107.465,Z 448.068,A -85,B 0,C 180,E1 -28411.991,E2 -28411.991} C_VEL
LIN {X 0,Y 117.578,Z 439.359,A -85,B 0,C 180,E1 -28415.72,E2 -28415.72} C_VEL
LIN {X 0,Y 128.188,Z 428.882,A -85,B 0,C 180,E1 -28418.755,E2 -28418.755} C_VEL
LIN {X 0,Y 137.519,Z 418.119,A -85,B 0,C 180,E1 -28420.99,E2 -28420.99} C_VEL
LIN {X 0,Y 146.239,Z 406.367,A -85,B 0,C 180,E1 -28422.777,E2 -28422.777} C_VEL
LIN {X 0,Y 154.251,Z 393.532,A -85,B 0,C 180,E1 -28424.261,E2 -28424.261} C_VEL
LIN {X 0,Y 161.513,Z 379.36,A -85,B 0,C 180,E1 -28425.508,E2 -28425.508} C_VEL
LIN {X 0,Y 167.252,Z 365.534,A -85,B 0,C 180,E1 -28426.344,E2 -28426.344} C_VEL
LIN {X 0,Y 171.971,Z 350.806,A -85,B 0,C 180,E1 -28427.017,E2 -28427.017} C_VEL
LIN {X 0,Y 175.387,Z 336.083,A -85,B 0,C 180,E1 -28427.486,E2 -28427.486} C_VEL
LIN {X 0,Y 177.878,Z 318.754,A -85,B 0,C 180,E1 -28427.855,E2 -28427.855} C_VEL
LIN {X 0,Y 179.044,Z 308,A -85,B 0,C 180,E1 -28428.134,E2 -28428.134} C_VEL
LIN {X 0,Y 177.632,Z 303.886,A -85,B 0,C 180,E1 -28431.61,E2 -28431.61} C_VEL
LIN {X 0,Y 176.874,Z 301.478,A -85,B 0,C 180,E1 -28434.413,E2 -28434.413} C_VEL
LIN {X 0,Y 176.407,Z 298.597,A -85,B 0,C 180,E1 -28439.429,E2 -28439.429} C_VEL
LIN {X 0,Y 176.407,Z 298.845,A -85,B 0,C 180,E1 -28441.141,E2 -28441.141} C_VEL
LIN {X 0,Y 177.203,Z 302.437,A -85,B 0,C 180,E1 -28446.833,E2 -28446.833} C_VEL
LIN {X 0,Y 178.246,Z 305.617,A -85,B 0,C 180,E1 -28449.956,E2 -28449.956} C_VEL
LIN {X 0,Y 179.055,Z 307.939,A -85,B 0,C 180,E1 -28451.785,E2 -28451.785} C_VEL
LIN {X 0,Y 177.648,Z 320.841,A -85,B 0,C 180,E1 -28452.106,E2 -28452.106} C_VEL
LIN {X 0,Y 175.163,Z 337.559,A -85,B 0,C 180,E1 -28452.454,E2 -28452.454} C_VEL
LIN {X 0,Y 171.503,Z 352.945,A -85,B 0,C 180,E1 -28452.959,E2 -28452.959} C_VEL
LIN {X 0,Y 166.744,Z 367.319,A -85,B 0,C 180,E1 -28453.578,E2 -28453.578} C_VEL
LIN {X 0,Y 160.573,Z 381.814,A -85,B 0,C 180,E1 -28454.447,E2 -28454.447} C_VEL
LIN {X 0,Y 154.075,Z 394.255,A -85,B 0,C 180,E1 -28455.506,E2 -28455.506} C_VEL
LIN {X 0,Y 146.046,Z 407.126,A -85,B 0,C 180,E1 -28456.976,E2 -28456.976} C_VEL
LIN {X 0,Y 137.308,Z 418.911,A -85,B 0,C 180,E1 -28458.753,E2 -28458.753} C_VEL
LIN {X 0,Y 127.916,Z 429.71,A -85,B 0,C 180,E1 -28460.928,E2 -28460.928} C_VEL
LIN {X 0,Y 117.254,Z 440.226,A -85,B 0,C 180,E1 -28463.927,E2 -28463.927} C_VEL
LIN {X 0,Y 107.743,Z 448.449,A -85,B 0,C 180,E1 -28467.338,E2 -28467.338} C_VEL
LIN {X 0,Y 98.758,Z 455.32,A -85,B 0,C 180,E1 -28471.353,E2 -28471.353} C_VEL
LIN {X 0,Y 88.314,Z 462.272,A -85,B 0,C 180,E1 -28477.269,E2 -28477.269} C_VEL
LIN {X 0,Y 79.131,Z 467.739,A -85,B 0,C 180,E1 -28484.723,E2 -28484.723} C_VEL
LIN {X 0,Y 71.565,Z 471.872,A -85,B 0,C 180,E1 -28493.897,E2 -28493.897} C_VEL
LIN {X 0,Y 66.004,Z 474.769,A -85,B 0,C 180,E1 -28504.791,E2 -28504.791} C_VEL
LIN {X 0,Y 63.045,Z 476.497,A -85,B 0,C 180,E1 -28517.117,E2 -28517.117} C_VEL
LIN {X 0,Y 62.488,Z 477.088,A -85,B 0,C 180,E1 -28530,E2 -28530} C_VEL
LIN {X 0,Y 63.044,Z 476.475,A -85,B 0,C 180,E1 -28542.882,E2 -28542.882} C_VEL
LIN {X 0,Y 65.993,Z 474.717,A -85,B 0,C 180,E1 -28555.213,E2 -28555.213} C_VEL
LIN {X 0,Y 71.545,Z 471.794,A -85,B 0,C 180,E1 -28566.114,E2 -28566.114} C_VEL
LIN {X 0,Y 79.108,Z 467.637,A -85,B 0,C 180,E1 -28575.294,E2 -28575.294} C_VEL
LIN {X 0,Y 88.303,Z 462.135,A -85,B 0,C 180,E1 -28582.74,E2 -28582.74} C_VEL
LIN {X 0,Y 98.75,Z 455.14,A -85,B 0,C 180,E1 -28588.653,E2 -28588.653} C_VEL
LIN {X 0,Y 108.03,Z 447.952,A -85,B 0,C 180,E1 -28592.91,E2 -28592.91} C_VEL
LIN {X 0,Y 118.761,Z 438.637,A -85,B 0,C 180,E1 -28596.528,E2 -28596.528} C_VEL
LIN {X 0,Y 129.448,Z 427.789,A -85,B 0,C 180,E1 -28599.478,E2 -28599.478} C_VEL
LIN {X 0,Y 138.871,Z 416.621,A -85,B 0,C 180,E1 -28601.605,E2 -28601.605} C_VEL
LIN {X 0,Y 147.74,Z 404.223,A -85,B 0,C 180,E1 -28603.359,E2 -28603.359} C_VEL
LIN {X 0,Y 155.685,Z 390.898,A -85,B 0,C 180,E1 -28604.779,E2 -28604.779} C_VEL
LIN {X 0,Y 156.775,Z 388.817,A -85,B 0,C 180,E1 -28604.953,E2 -28604.953} C_VEL
LIN {X 0,Y 159.219,Z 383.725,A -85,B 0,C 180,E1 -28605.6,E2 -28605.6} C_VEL
LIN {X 0,Y 164.686,Z 368.628,A -85,B 0,C 180,E1 -28608.365,E2 -28608.365} C_VEL
LIN {X 0,Y 166.444,Z 363.264,A -85,B 0,C 180,E1 -28608.957,E2 -28608.957} C_VEL
LIN {X 0,Y 167.049,Z 361.417,A -85,B 0,C 180,E1 -28609.059,E2 -28609.059} C_VEL
LIN {X 0,Y 171.511,Z 346.397,A -85,B 0,C 180,E1 -28609.56,E2 -28609.56} C_VEL
LIN {X 0,Y 174.702,Z 330.599,A -85,B 0,C 180,E1 -28609.945,E2 -28609.945} C_VEL
LIN {X 0,Y 176.925,Z 312.518,A -85,B 0,C 180,E1 -28610.297,E2 -28610.297} C_VEL
LIN {X 0,Y 175.824,Z 308.69,A -85,B 0,C 180,E1 -28613.957,E2 -28613.957} C_VEL
LIN {X 0,Y 175.224,Z 305.477,A -85,B 0,C 180,E1 -28619.426,E2 -28619.426} C_VEL
LIN {X 0,Y 175.228,Z 305.592,A -85,B 0,C 180,E1 -28621.149,E2 -28621.149} C_VEL
LIN {X 0,Y 175.894,Z 309.161,A -85,B 0,C 180,E1 -28626.597,E2 -28626.597} C_VEL
LIN {X 0,Y 176.896,Z 312.535,A -85,B 0,C 180,E1 -28629.829,E2 -28629.829} C_VEL
LIN {X 0,Y 174.125,Z 333.717,A -85,B 0,C 180,E1 -28630.299,E2 -28630.299} C_VEL
LIN {X 0,Y 170.677,Z 349.133,A -85,B 0,C 180,E1 -28630.697,E2 -28630.697} C_VEL
LIN {X 0,Y 166.155,Z 363.571,A -85,B 0,C 180,E1 -28631.282,E2 -28631.282} C_VEL
LIN {X 0,Y 160.756,Z 376.907,A -85,B 0,C 180,E1 -28631.985,E2 -28631.985} C_VEL
LIN {X 0,Y 154.15,Z 390.144,A -85,B 0,C 180,E1 -28632.96,E2 -28632.96} C_VEL
LIN {X 0,Y 146.419,Z 402.965,A -85,B 0,C 180,E1 -28634.268,E2 -28634.268} C_VEL
LIN {X 0,Y 137.029,Z 415.824,A -85,B 0,C 180,E1 -28635.918,E2 -28635.918} C_VEL
LIN {X 0,Y 127.407,Z 426.967,A -85,B 0,C 180,E1 -28637.91,E2 -28637.91} C_VEL
LIN {X 0,Y 116.415,Z 437.784,A -85,B 0,C 180,E1 -28640.653,E2 -28640.653} C_VEL
LIN {X 0,Y 105.807,Z 446.771,A -85,B 0,C 180,E1 -28644.033,E2 -28644.033} C_VEL
LIN {X 0,Y 95.571,Z 454.218,A -85,B 0,C 180,E1 -28648.062,E2 -28648.062} C_VEL
LIN {X 0,Y 84.628,Z 461.177,A -85,B 0,C 180,E1 -28653.855,E2 -28653.855} C_VEL
LIN {X 0,Y 74.28,Z 466.845,A -85,B 0,C 180,E1 -28661.477,E2 -28661.477} C_VEL
LIN {X 0,Y 66.354,Z 470.764,A -85,B 0,C 180,E1 -28670.543,E2 -28670.543} C_VEL
LIN {X 0,Y 59.994,Z 473.656,A -85,B 0,C 180,E1 -28682.058,E2 -28682.058} C_VEL
LIN {X 0,Y 56.32,Z 475.388,A -85,B 0,C 180,E1 -28695.548,E2 -28695.548} C_VEL
LIN {X 0,Y 55.465,Z 475.985,A -85,B 0,C 180,E1 -28710,E2 -28710} C_VEL
LIN {X 0,Y 56.312,Z 475.416,A -85,B 0,C 180,E1 -28724.455,E2 -28724.455} C_VEL
LIN {X 0,Y 59.946,Z 473.723,A -85,B 0,C 180,E1 -28737.967,E2 -28737.967} C_VEL
LIN {X 0,Y 66.341,Z 470.864,A -85,B 0,C 180,E1 -28749.467,E2 -28749.467} C_VEL
LIN {X 0,Y 74.683,Z 466.774,A -85,B 0,C 180,E1 -28758.837,E2 -28758.837} C_VEL
LIN {X 0,Y 84.579,Z 461.351,A -85,B 0,C 180,E1 -28766.196,E2 -28766.196} C_VEL
LIN {X 0,Y 95.54,Z 454.441,A -85,B 0,C 180,E1 -28771.975,E2 -28771.975} C_VEL
LIN {X 0,Y 104.29,Z 448.134,A -85,B 0,C 180,E1 -28775.472,E2 -28775.472} C_VEL
LIN {X 0,Y 114.822,Z 439.423,A -85,B 0,C 180,E1 -28778.974,E2 -28778.974} C_VEL
LIN {X 0,Y 125.783,Z 428.946,A -85,B 0,C 180,E1 -28781.78,E2 -28781.78} C_VEL
LIN {X 0,Y 135.371,Z 418.182,A -85,B 0,C 180,E1 -28783.835,E2 -28783.835} C_VEL
LIN {X 0,Y 144.297,Z 406.43,A -85,B 0,C 180,E1 -28785.471,E2 -28785.471} C_VEL
LIN {X 0,Y 152.475,Z 393.594,A -85,B 0,C 180,E1 -28786.835,E2 -28786.835} C_VEL
LIN {X 0,Y 159.884,Z 379.421,A -85,B 0,C 180,E1 -28787.971,E2 -28787.971} C_VEL
LIN {X 0,Y 165.72,Z 365.593,A -85,B 0,C 180,E1 -28788.728,E2 -28788.728} C_VEL
LIN {X 0,Y 170.518,Z 350.863,A -85,B 0,C 180,E1 -28789.339,E2 -28789.339} C_VEL
LIN {X 0,Y 174.025,Z 335.943,A -85,B 0,C 180,E1 -28789.767,E2 -28789.767} C_VEL
LIN {X 0,Y 176.523,Z 318.79,A -85,B 0,C 180,E1 -28790.107,E2 -28790.107} C_VEL
LIN {X 0,Y 177.175,Z 312.754,A -85,B 0,C 180,E1 -28790.294,E2 -28790.294} C_VEL
LIN {X 0,Y 176.271,Z 309.823,A -85,B 0,C 180,E1 -28793.13,E2 -28793.13} C_VEL
LIN {X 0,Y 175.908,Z 308.415,A -85,B 0,C 180,E1 -28794.796,E2 -28794.796} C_VEL
LIN {X 0,Y 175.538,Z 305.681,A -85,B 0,C 180,E1 -28799.426,E2 -28799.426} C_VEL
LIN {X 0,Y 175.529,Z 305.871,A -85,B 0,C 180,E1 -28800.86,E2 -28800.86} C_VEL
LIN {X 0,Y 176.15,Z 309.206,A -85,B 0,C 180,E1 -28806.224,E2 -28806.224} C_VEL
LIN {X 0,Y 177.007,Z 312.119,A -85,B 0,C 180,E1 -28809.138,E2 -28809.138} C_VEL
LIN {X 0,Y 177.209,Z 312.811,A -85,B 0,C 180,E1 -28809.697,E2 -28809.697} C_VEL
LIN {X 0,Y 174.448,Z 333.82,A -85,B 0,C 180,E1 -28810.085,E2 -28810.085} C_VEL
LIN {X 0,Y 171.109,Z 349.054,A -85,B 0,C 180,E1 -28810.507,E2 -28810.507} C_VEL
LIN {X 0,Y 166.478,Z 363.869,A -85,B 0,C 180,E1 -28811.032,E2 -28811.032} C_VEL
LIN {X 0,Y 160.617,Z 378.22,A -85,B 0,C 180,E1 -28811.749,E2 -28811.749} C_VEL
LIN {X 0,Y 153.975,Z 391.341,A -85,B 0,C 180,E1 -28812.673,E2 -28812.673} C_VEL
LIN {X 0,Y 146.112,Z 404.2,A -85,B 0,C 180,E1 -28813.916,E2 -28813.916} C_VEL
LIN {X 0,Y 137.619,Z 415.891,A -85,B 0,C 180,E1 -28815.437,E2 -28815.437} C_VEL
LIN {X 0,Y 127.133,Z 428.016,A -85,B 0,C 180,E1 -28817.523,E2 -28817.523} C_VEL
LIN {X 0,Y 116.1,Z 438.806,A -85,B 0,C 180,E1 -28820.234,E2 -28820.234} C_VEL
LIN {X 0,Y 105.27,Z 447.909,A -85,B 0,C 180,E1 -28823.613,E2 -28823.613} C_VEL
LIN {X 0,Y 95.235,Z 455.254,A -85,B 0,C 180,E1 -28827.679,E2 -28827.679} C_VEL
LIN {X 0,Y 84.169,Z 462.206,A -85,B 0,C 180,E1 -28833.385,E2 -28833.385} C_VEL
LIN {X 0,Y 74.27,Z 467.673,A -85,B 0,C 180,E1 -28840.797,E2 -28840.797} C_VEL
LIN {X 0,Y 65.911,Z 471.806,A -85,B 0,C 180,E1 -28850.225,E2 -28850.225} C_VEL
LIN {X 0,Y 59.607,Z 474.702,A -85,B 0,C 180,E1 -28861.86,E2 -28861.86} C_VEL
LIN {X 0,Y 56.105,Z 476.431,A -85,B 0,C 180,E1 -28875.491,E2 -28875.491} C_VEL
LIN {X 0,Y 55.387,Z 477.022,A -85,B 0,C 180,E1 -28890,E2 -28890} C_VEL
LIN {X 0,Y 56.104,Z 476.408,A -85,B 0,C 180,E1 -28904.509,E2 -28904.509} C_VEL
LIN {X 0,Y 59.595,Z 474.649,A -85,B 0,C 180,E1 -28918.146,E2 -28918.146} C_VEL
LIN {X 0,Y 65.891,Z 471.727,A -85,B 0,C 180,E1 -28929.789,E2 -28929.789} C_VEL
LIN {X 0,Y 74.236,Z 467.569,A -85,B 0,C 180,E1 -28939.233,E2 -28939.233} C_VEL
LIN {X 0,Y 84.162,Z 462.067,A -85,B 0,C 180,E1 -28946.621,E2 -28946.621} C_VEL
LIN {X 0,Y 95.226,Z 455.072,A -85,B 0,C 180,E1 -28952.33,E2 -28952.33} C_VEL
LIN {X 0,Y 104.975,Z 447.88,A -85,B 0,C 180,E1 -28956.386,E2 -28956.386} C_VEL
LIN {X 0,Y 116.104,Z 438.568,A -85,B 0,C 180,E1 -28959.759,E2 -28959.759} C_VEL
LIN {X 0,Y 127.121,Z 427.72,A -85,B 0,C 180,E1 -28962.493,E2 -28962.493} C_VEL
LIN {X 0,Y 136.796,Z 416.551,A -85,B 0,C 180,E1 -28964.428,E2 -28964.428} C_VEL
LIN {X 0,Y 144.937,Z 405.478,A -85,B 0,C 180,E1 -28965.884,E2 -28965.884} C_VEL
LIN {X 0,Y 153.147,Z 392.256,A -85,B 0,C 180,E1 -28967.207,E2 -28967.207} C_VEL
LIN {X 0,Y 159.785,Z 379.343,A -85,B 0,C 180,E1 -28968.139,E2 -28968.139} C_VEL
LIN {X 0,Y 165.629,Z 365.32,A -85,B 0,C 180,E1 -28968.886,E2 -28968.886} C_VEL
LIN {X 0,Y 167.049,Z 361.417,A -85,B 0,C 180,E1 -28969.059,E2 -28969.059} C_VEL
LIN {X 0,Y 168.738,Z 355.873,A -85,B 0,C 180,E1 -28969.47,E2 -28969.47} C_VEL
LIN {X 0,Y 170.785,Z 346.872,A -85,B 0,C 180,E1 -28970.7,E2 -28970.7} C_VEL
LIN {X 0,Y 172.393,Z 337.756,A -85,B 0,C 180,E1 -28971.884,E2 -28971.884} C_VEL
LIN {X 0,Y 173.354,Z 332.03,A -85,B 0,C 180,E1 -28972.229,E2 -28972.229} C_VEL
LIN {X 0,Y 175.272,Z 317.455,A -85,B 0,C 180,E1 -28972.512,E2 -28972.512} C_VEL
LIN {X 0,Y 174.681,Z 315.201,A -85,B 0,C 180,E1 -28975.096,E2 -28975.096} C_VEL
LIN {X 0,Y 174.359,Z 312.51,A -85,B 0,C 180,E1 -28979.466,E2 -28979.466} C_VEL
LIN {X 0,Y 174.345,Z 312.731,A -85,B 0,C 180,E1 -28981.028,E2 -28981.028} C_VEL
LIN {X 0,Y 174.892,Z 316.089,A -85,B 0,C 180,E1 -28986.164,E2 -28986.164} C_VEL
LIN {X 0,Y 175.267,Z 317.499,A -85,B 0,C 180,E1 -28987.667,E2 -28987.667} C_VEL
LIN {X 0,Y 172.852,Z 334.598,A -85,B 0,C 180,E1 -28988.008,E2 -28988.008} C_VEL
LIN {X 0,Y 169.32,Z 349.867,A -85,B 0,C 180,E1 -28988.361,E2 -28988.361} C_VEL
LIN {X 0,Y 164.421,Z 364.943,A -85,B 0,C 180,E1 -28988.906,E2 -28988.906} C_VEL
LIN {X 0,Y 158.589,Z 378.743,A -85,B 0,C 180,E1 -28989.589,E2 -28989.589} C_VEL
LIN {X 0,Y 151.877,Z 391.641,A -85,B 0,C 180,E1 -28990.477,E2 -28990.477} C_VEL
LIN {X 0,Y 143.559,Z 404.841,A -85,B 0,C 180,E1 -28991.733,E2 -28991.733} C_VEL
LIN {X 0,Y 135.254,Z 415.894,A -85,B 0,C 180,E1 -28993.024,E2 -28993.024} C_VEL
LIN {X 0,Y 125.403,Z 427.036,A -85,B 0,C 180,E1 -28994.818,E2 -28994.818} C_VEL
LIN {X 0,Y 114.096,Z 437.853,A -85,B 0,C 180,E1 -28997.301,E2 -28997.301} C_VEL
LIN {X 0,Y 103.092,Z 446.84,A -85,B 0,C 180,E1 -29000.387,E2 -29000.387} C_VEL
LIN {X 0,Y 92.435,Z 454.286,A -85,B 0,C 180,E1 -29004.163,E2 -29004.163} C_VEL
LIN {X 0,Y 80.866,Z 461.245,A -85,B 0,C 180,E1 -29009.646,E2 -29009.646} C_VEL
LIN {X 0,Y 69.107,Z 467.23,A -85,B 0,C 180,E1 -29017.604,E2 -29017.604} C_VEL
LIN {X 0,Y 61.002,Z 470.832,A -85,B 0,C 180,E1 -29026.271,E2 -29026.271} C_VEL
LIN {X 0,Y 53.779,Z 473.723,A -85,B 0,C 180,E1 -29038.485,E2 -29038.485} C_VEL
LIN {X 0,Y 49.468,Z 475.454,A -85,B 0,C 180,E1 -29053.493,E2 -29053.493} C_VEL
LIN {X 0,Y 48.366,Z 476.052,A -85,B 0,C 180,E1 -29070,E2 -29070} C_VEL
LIN {X 0,Y 49.46,Z 475.483,A -85,B 0,C 180,E1 -29086.511,E2 -29086.511} C_VEL
LIN {X 0,Y 53.735,Z 473.789,A -85,B 0,C 180,E1 -29101.545,E2 -29101.545} C_VEL
LIN {X 0,Y 60.992,Z 470.93,A -85,B 0,C 180,E1 -29113.739,E2 -29113.739} C_VEL
LIN {X 0,Y 70.188,Z 466.839,A -85,B 0,C 180,E1 -29123.231,E2 -29123.231} C_VEL
LIN {X 0,Y 80.819,Z 461.416,A -85,B 0,C 180,E1 -29130.412,E2 -29130.412} C_VEL
LIN {X 0,Y 92.41,Z 454.506,A -85,B 0,C 180,E1 -29135.872,E2 -29135.872} C_VEL
LIN {X 0,Y 103.044,Z 447.086,A -85,B 0,C 180,E1 -29139.686,E2 -29139.686} C_VEL
LIN {X 0,Y 114.061,Z 438.137,A -85,B 0,C 180,E1 -29142.758,E2 -29142.758} C_VEL
LIN {X 0,Y 125.359,Z 427.386,A -85,B 0,C 180,E1 -29145.26,E2 -29145.26} C_VEL
LIN {X 0,Y 136.037,Z 415.298,A -85,B 0,C 180,E1 -29147.196,E2 -29147.196} C_VEL
LIN {X 0,Y 145.546,Z 402.383,A -85,B 0,C 180,E1 -29148.673,E2 -29148.673} C_VEL
LIN {X 0,Y 153.523,Z 389.328,A -85,B 0,C 180,E1 -29149.812,E2 -29149.812} C_VEL
LIN {X 0,Y 160.243,Z 375.938,A -85,B 0,C 180,E1 -29150.687,E2 -29150.687} C_VEL
LIN {X 0,Y 166.038,Z 361.465,A -85,B 0,C 180,E1 -29151.346,E2 -29151.346} C_VEL
LIN {X 0,Y 170.673,Z 346.115,A -85,B 0,C 180,E1 -29151.848,E2 -29151.848} C_VEL
LIN {X 0,Y 173.964,Z 330.149,A -85,B 0,C 180,E1 -29152.189,E2 -29152.189} C_VEL
LIN {X 0,Y 175.557,Z 317.712,A -85,B 0,C 180,E1 -29152.452,E2 -29152.452} C_VEL
LIN {X 0,Y 174.91,Z 315.256,A -85,B 0,C 180,E1 -29155.39,E2 -29155.39} C_VEL
LIN {X 0,Y 174.678,Z 312.619,A -85,B 0,C 180,E1 -29160,E2 -29160} C_VEL
LIN {X 0,Y 175.146,Z 316.113,A -85,B 0,C 180,E1 -29165.757,E2 -29165.757} C_VEL
LIN {X 0,Y 175.572,Z 317.671,A -85,B 0,C 180,E1 -29167.487,E2 -29167.487} C_VEL
LIN {X 0,Y 173.117,Z 334.999,A -85,B 0,C 180,E1 -29167.801,E2 -29167.801} C_VEL
LIN {X 0,Y 169.601,Z 350.284,A -85,B 0,C 180,E1 -29168.194,E2 -29168.194} C_VEL
LIN {X 0,Y 164.785,Z 365.093,A -85,B 0,C 180,E1 -29168.668,E2 -29168.668} C_VEL
LIN {X 0,Y 158.476,Z 379.926,A -85,B 0,C 180,E1 -29169.344,E2 -29169.344} C_VEL
LIN {X 0,Y 151.731,Z 392.705,A -85,B 0,C 180,E1 -29170.174,E2 -29170.174} C_VEL
LIN {X 0,Y 143.369,Z 405.825,A -85,B 0,C 180,E1 -29171.36,E2 -29171.36} C_VEL
LIN {X 0,Y 135.067,Z 416.83,A -85,B 0,C 180,E1 -29172.675,E2 -29172.675} C_VEL
LIN {X 0,Y 125.167,Z 427.952,A -85,B 0,C 180,E1 -29174.402,E2 -29174.402} C_VEL
LIN {X 0,Y 113.829,Z 438.741,A -85,B 0,C 180,E1 -29176.863,E2 -29176.863} C_VEL
LIN {X 0,Y 104.331,Z 446.521,A -85,B 0,C 180,E1 -29179.424,E2 -29179.424} C_VEL
LIN {X 0,Y 92.133,Z 455.189,A -85,B 0,C 180,E1 -29183.741,E2 -29183.741} C_VEL
LIN {X 0,Y 80.455,Z 462.141,A -85,B 0,C 180,E1 -29189.128,E2 -29189.128} C_VEL
LIN {X 0,Y 69.807,Z 467.607,A -85,B 0,C 180,E1 -29196.348,E2 -29196.348} C_VEL
LIN {X 0,Y 60.58,Z 471.74,A -85,B 0,C 180,E1 -29205.887,E2 -29205.887} C_VEL
LIN {X 0,Y 53.403,Z 474.636,A -85,B 0,C 180,E1 -29218.236,E2 -29218.236} C_VEL
LIN {X 0,Y 49.235,Z 476.364,A -85,B 0,C 180,E1 -29233.412,E2 -29233.412} C_VEL
LIN {X 0,Y 48.302,Z 476.955,A -85,B 0,C 180,E1 -29250,E2 -29250} C_VEL
LIN {X 0,Y 49.234,Z 476.341,A -85,B 0,C 180,E1 -29266.588,E2 -29266.588} C_VEL
LIN {X 0,Y 53.39,Z 474.582,A -85,B 0,C 180,E1 -29281.772,E2 -29281.772} C_VEL
LIN {X 0,Y 60.56,Z 471.659,A -85,B 0,C 180,E1 -29294.131,E2 -29294.131} C_VEL
LIN {X 0,Y 69.765,Z 467.501,A -85,B 0,C 180,E1 -29303.698,E2 -29303.698} C_VEL
LIN {X 0,Y 80.451,Z 461.999,A -85,B 0,C 180,E1 -29310.877,E2 -29310.877} C_VEL
LIN {X 0,Y 92.122,Z 455.003,A -85,B 0,C 180,E1 -29316.274,E2 -29316.274} C_VEL
LIN {X 0,Y 101.979,Z 448.06,A -85,B 0,C 180,E1 -29319.942,E2 -29319.942} C_VEL
LIN {X 0,Y 113.834,Z 438.499,A -85,B 0,C 180,E1 -29323.128,E2 -29323.128} C_VEL
LIN {X 0,Y 125.156,Z 427.65,A -85,B 0,C 180,E1 -29325.617,E2 -29325.617} C_VEL
LIN {X 0,Y 135.062,Z 416.482,A -85,B 0,C 180,E1 -29327.333,E2 -29327.333} C_VEL
LIN {X 0,Y 144.117,Z 404.353,A -85,B 0,C 180,E1 -29328.752,E2 -29328.752} C_VEL
LIN {X 0,Y 152.569,Z 390.756,A -85,B 0,C 180,E1 -29329.94,E2 -29329.94} C_VEL
LIN {X 0,Y 159.317,Z 377.504,A -85,B 0,C 180,E1 -29330.763,E2 -29330.763} C_VEL
LIN {X 0,Y 165.499,Z 362.344,A -85,B 0,C 180,E1 -29331.432,E2 -29331.432} C_VEL
LIN {X 0,Y 170.201,Z 346.986,A -85,B 0,C 180,E1 -29331.892,E2 -29331.892} C_VEL
LIN {X 0,Y 173.354,Z 332.03,A -85,B 0,C 180,E1 -29332.229,E2 -29332.229} C_VEL
LIN {X 0,Y 173.758,Z 329,A -85,B 0,C 180,E1 -29332.563,E2 -29332.563} C_VEL
LIN {X 0,Y 173.896,Z 326.02,A -85,B 0,C 180,E1 -29333.437,E2 -29333.437} C_VEL
LIN {X 0,Y 173.787,Z 323.51,A -85,B 0,C 180,E1 -29334.821,E2 -29334.821} C_VEL
LIN {X 0,Y 173.517,Z 321.174,A -85,B 0,C 180,E1 -29337.184,E2 -29337.184} C_VEL
LIN {X 0,Y 173.458,Z 320.563,A -85,B 0,C 180,E1 -29338.162,E2 -29338.162} C_VEL
LIN {X 0,Y 173.494,Z 319.472,A -85,B 0,C 180,E1 -29340,E2 -29340} C_VEL
LIN {X 0,Y 173.846,Z 322.768,A -85,B 0,C 180,E1 -29345.437,E2 -29345.437} C_VEL
LIN {X 0,Y 171.3,Z 338.424,A -85,B 0,C 180,E1 -29345.733,E2 -29345.733} C_VEL
LIN {X 0,Y 167.588,Z 352.971,A -85,B 0,C 180,E1 -29346.073,E2 -29346.073} C_VEL
LIN {X 0,Y 162.273,Z 368.18,A -85,B 0,C 180,E1 -29346.578,E2 -29346.578} C_VEL
LIN {X 0,Y 155.856,Z 382.342,A -85,B 0,C 180,E1 -29347.233,E2 -29347.233} C_VEL
LIN {X 0,Y 148.338,Z 395.763,A -85,B 0,C 180,E1 -29348.127,E2 -29348.127} C_VEL
LIN {X 0,Y 139.74,Z 408.427,A -85,B 0,C 180,E1 -29349.246,E2 -29349.246} C_VEL
LIN {X 0,Y 130.463,Z 419.859,A -85,B 0,C 180,E1 -29350.542,E2 -29350.542} C_VEL
LIN {X 0,Y 120.452,Z 430.362,A -85,B 0,C 180,E1 -29352.228,E2 -29352.228} C_VEL
LIN {X 0,Y 108.899,Z 440.623,A -85,B 0,C 180,E1 -29354.523,E2 -29354.523} C_VEL
LIN {X 0,Y 97.662,Z 449.139,A -85,B 0,C 180,E1 -29357.541,E2 -29357.541} C_VEL
LIN {X 0,Y 86.639,Z 456.228,A -85,B 0,C 180,E1 -29361.114,E2 -29361.114} C_VEL
LIN {X 0,Y 74.64,Z 462.803,A -85,B 0,C 180,E1 -29366.555,E2 -29366.555} C_VEL
LIN {X 0,Y 64.295,Z 467.599,A -85,B 0,C 180,E1 -29373.131,E2 -29373.131} C_VEL
LIN {X 0,Y 56.045,Z 470.9,A -85,B 0,C 180,E1 -29381.202,E2 -29381.202} C_VEL
LIN {X 0,Y 47.829,Z 473.791,A -85,B 0,C 180,E1 -29394.002,E2 -29394.002} C_VEL
LIN {X 0,Y 42.677,Z 475.521,A -85,B 0,C 180,E1 -29410.771,E2 -29410.771} C_VEL
LIN {X 0,Y 41.282,Z 476.118,A -85,B 0,C 180,E1 -29430,E2 -29430} C_VEL
LIN {X 0,Y 42.667,Z 475.549,A -85,B 0,C 180,E1 -29449.235,E2 -29449.235} C_VEL
LIN {X 0,Y 47.79,Z 473.856,A -85,B 0,C 180,E1 -29466.032,E2 -29466.032} C_VEL
LIN {X 0,Y 56.038,Z 470.996,A -85,B 0,C 180,E1 -29478.807,E2 -29478.807} C_VEL
LIN {X 0,Y 66.163,Z 466.905,A -85,B 0,C 180,E1 -29488.189,E2 -29488.189} C_VEL
LIN {X 0,Y 77.535,Z 461.482,A -85,B 0,C 180,E1 -29495.017,E2 -29495.017} C_VEL
LIN {X 0,Y 89.739,Z 454.571,A -85,B 0,C 180,E1 -29500.017,E2 -29500.017} C_VEL
LIN {X 0,Y 100.786,Z 447.151,A -85,B 0,C 180,E1 -29503.501,E2 -29503.501} C_VEL
LIN {X 0,Y 112.151,Z 438.201,A -85,B 0,C 180,E1 -29506.245,E2 -29506.245} C_VEL
LIN {X 0,Y 122.073,Z 429.075,A -85,B 0,C 180,E1 -29508.161,E2 -29508.161} C_VEL
LIN {X 0,Y 132.12,Z 418.309,A -85,B 0,C 180,E1 -29509.769,E2 -29509.769} C_VEL
LIN {X 0,Y 141.402,Z 406.555,A -85,B 0,C 180,E1 -29511.056,E2 -29511.056} C_VEL
LIN {X 0,Y 149.878,Z 393.718,A -85,B 0,C 180,E1 -29512.132,E2 -29512.132} C_VEL
LIN {X 0,Y 157.537,Z 379.542,A -85,B 0,C 180,E1 -29513.033,E2 -29513.033} C_VEL
LIN {X 0,Y 163.418,Z 366.032,A -85,B 0,C 180,E1 -29513.597,E2 -29513.597} C_VEL
LIN {X 0,Y 168.248,Z 351.767,A -85,B 0,C 180,E1 -29514.066,E2 -29514.066} C_VEL
LIN {X 0,Y 171.931,Z 336.788,A -85,B 0,C 180,E1 -29514.412,E2 -29514.412} C_VEL
LIN {X 0,Y 174.136,Z 323.048,A -85,B 0,C 180,E1 -29514.681,E2 -29514.681} C_VEL
LIN {X 0,Y 173.805,Z 321.399,A -85,B 0,C 180,E1 -29517.175,E2 -29517.175} C_VEL
LIN {X 0,Y 173.807,Z 319.716,A -85,B 0,C 180,E1 -29520,E2 -29520} C_VEL
LIN {X 0,Y 174.145,Z 322.996,A -85,B 0,C 180,E1 -29525.243,E2 -29525.243} C_VEL
LIN {X 0,Y 171.574,Z 338.79,A -85,B 0,C 180,E1 -29525.541,E2 -29525.541} C_VEL
LIN {X 0,Y 167.503,Z 354.538,A -85,B 0,C 180,E1 -29525.91,E2 -29525.91} C_VEL
LIN {X 0,Y 162.207,Z 369.364,A -85,B 0,C 180,E1 -29526.37,E2 -29526.37} C_VEL
LIN {X 0,Y 155.767,Z 383.387,A -85,B 0,C 180,E1 -29526.966,E2 -29526.966} C_VEL
LIN {X 0,Y 148.085,Z 396.916,A -85,B 0,C 180,E1 -29527.814,E2 -29527.814} C_VEL
LIN {X 0,Y 139.426,Z 409.528,A -85,B 0,C 180,E1 -29528.91,E2 -29528.91} C_VEL
LIN {X 0,Y 130.313,Z 420.675,A -85,B 0,C 180,E1 -29530.18,E2 -29530.18} C_VEL
LIN {X 0,Y 120.253,Z 431.147,A -85,B 0,C 180,E1 -29531.782,E2 -29531.782} C_VEL
LIN {X 0,Y 108.677,Z 441.388,A -85,B 0,C 180,E1 -29534.062,E2 -29534.062} C_VEL
LIN {X 0,Y 97.613,Z 449.73,A -85,B 0,C 180,E1 -29536.912,E2 -29536.912} C_VEL
LIN {X 0,Y 86.376,Z 456.985,A -85,B 0,C 180,E1 -29540.658,E2 -29540.658} C_VEL
LIN {X 0,Y 74.274,Z 463.555,A -85,B 0,C 180,E1 -29545.984,E2 -29545.984} C_VEL
LIN {X 0,Y 65.816,Z 467.541,A -85,B 0,C 180,E1 -29551.321,E2 -29551.321} C_VEL
LIN {X 0,Y 55.665,Z 471.673,A -85,B 0,C 180,E1 -29560.752,E2 -29560.752} C_VEL
LIN {X 0,Y 47.471,Z 474.57,A -85,B 0,C 180,E1 -29573.687,E2 -29573.687} C_VEL
LIN {X 0,Y 42.433,Z 476.298,A -85,B 0,C 180,E1 -29590.655,E2 -29590.655} C_VEL
LIN {X 0,Y 41.187,Z 476.889,A -85,B 0,C 180,E1 -29610,E2 -29610} C_VEL
LIN {X 0,Y 42.431,Z 476.274,A -85,B 0,C 180,E1 -29629.345,E2 -29629.345} C_VEL
LIN {X 0,Y 47.459,Z 474.515,A -85,B 0,C 180,E1 -29646.323,E2 -29646.323} C_VEL
LIN {X 0,Y 55.643,Z 471.591,A -85,B 0,C 180,E1 -29659.273,E2 -29659.273} C_VEL
LIN {X 0,Y 65.771,Z 467.433,A -85,B 0,C 180,E1 -29668.742,E2 -29668.742} C_VEL
LIN {X 0,Y 77.22,Z 461.931,A -85,B 0,C 180,E1 -29675.523,E2 -29675.523} C_VEL
LIN {X 0,Y 89.48,Z 454.935,A -85,B 0,C 180,E1 -29680.478,E2 -29680.478} C_VEL
LIN {X 0,Y 100.759,Z 447.282,A -85,B 0,C 180,E1 -29684.063,E2 -29684.063} C_VEL
LIN {X 0,Y 111.975,Z 438.431,A -85,B 0,C 180,E1 -29686.617,E2 -29686.617} C_VEL
LIN {X 0,Y 123.578,Z 427.581,A -85,B 0,C 180,E1 -29688.82,E2 -29688.82} C_VEL
LIN {X 0,Y 133.683,Z 416.412,A -85,B 0,C 180,E1 -29690.308,E2 -29690.308} C_VEL
LIN {X 0,Y 143.661,Z 403.187,A -85,B 0,C 180,E1 -29691.655,E2 -29691.655} C_VEL
LIN {X 0,Y 151.488,Z 390.685,A -85,B 0,C 180,E1 -29692.593,E2 -29692.593} C_VEL
LIN {X 0,Y 158.331,Z 377.432,A -85,B 0,C 180,E1 -29693.304,E2 -29693.304} C_VEL
LIN {X 0,Y 164.037,Z 363.723,A -85,B 0,C 180,E1 -29693.83,E2 -29693.83} C_VEL
LIN {X 0,Y 168.653,Z 349.372,A -85,B 0,C 180,E1 -29694.207,E2 -29694.207} C_VEL
LIN {X 0,Y 172.207,Z 333.721,A -85,B 0,C 180,E1 -29694.533,E2 -29694.533} C_VEL
LIN {X 0,Y 173.852,Z 322.627,A -85,B 0,C 180,E1 -29694.782,E2 -29694.782} C_VEL
LIN {X 0,Y 173.458,Z 320.563,A -85,B 0,C 180,E1 -29698.162,E2 -29698.162} C_VEL
LIN {X 0,Y 173.353,Z 320.944,A -85,B 0,C 180,E1 -29698.935,E2 -29698.935} C_VEL
LIN {X 0,Y 172.996,Z 323.518,A -85,B 0,C 180,E1 -29700.029,E2 -29700.029} C_VEL
LIN {X 0,Y 172.579,Z 326.607,A -85,B 0,C 180,E1 -29701.112,E2 -29701.112} C_VEL
LIN {X 0,Y 172.477,Z 327.677,A -85,B 0,C 180,E1 -29701.904,E2 -29701.904} C_VEL
LIN {X 0,Y 172.533,Z 328.426,A -85,B 0,C 180,E1 -29703.19,E2 -29703.19} C_VEL
LIN {X 0,Y 169.625,Z 343.242,A -85,B 0,C 180,E1 -29703.437,E2 -29703.437} C_VEL
LIN {X 0,Y 165.165,Z 358.645,A -85,B 0,C 180,E1 -29703.798,E2 -29703.798} C_VEL
LIN {X 0,Y 159.446,Z 373.286,A -85,B 0,C 180,E1 -29704.246,E2 -29704.246} C_VEL
LIN {X 0,Y 152.532,Z 387.232,A -85,B 0,C 180,E1 -29704.875,E2 -29704.875} C_VEL
LIN {X 0,Y 144.784,Z 400.005,A -85,B 0,C 180,E1 -29705.706,E2 -29705.706} C_VEL
LIN {X 0,Y 135.348,Z 412.864,A -85,B 0,C 180,E1 -29706.746,E2 -29706.746} C_VEL
LIN {X 0,Y 125.941,Z 423.627,A -85,B 0,C 180,E1 -29707.894,E2 -29707.894} C_VEL
LIN {X 0,Y 115.759,Z 433.58,A -85,B 0,C 180,E1 -29709.399,E2 -29709.399} C_VEL
LIN {X 0,Y 103.991,Z 443.307,A -85,B 0,C 180,E1 -29711.502,E2 -29711.502} C_VEL
LIN {X 0,Y 92.476,Z 451.408,A -85,B 0,C 180,E1 -29714.31,E2 -29714.31} C_VEL
LIN {X 0,Y 81.13,Z 458.1,A -85,B 0,C 180,E1 -29717.658,E2 -29717.658} C_VEL
LIN {X 0,Y 68.665,Z 464.29,A -85,B 0,C 180,E1 -29722.902,E2 -29722.902} C_VEL
LIN {X 0,Y 56.976,Z 469.067,A -85,B 0,C 180,E1 -29730.294,E2 -29730.294} C_VEL
LIN {X 0,Y 46.654,Z 472.561,A -85,B 0,C 180,E1 -29741.131,E2 -29741.131} C_VEL
LIN {X 0,Y 38.676,Z 474.865,A -85,B 0,C 180,E1 -29756.966,E2 -29756.966} C_VEL
LIN {X 0,Y 34.493,Z 476.031,A -85,B 0,C 180,E1 -29778.244,E2 -29778.244} C_VEL
LIN {X 0,Y 34.171,Z 476.184,A -85,B 0,C 180,E1 -29790.001,E2 -29790.001} C_VEL
LIN {X 0,Y 36.016,Z 475.615,A -85,B 0,C 180,E1 -29812.972,E2 -29812.972} C_VEL
LIN {X 0,Y 42.222,Z 473.922,A -85,B 0,C 180,E1 -29831.745,E2 -29831.745} C_VEL
LIN {X 0,Y 51.605,Z 471.062,A -85,B 0,C 180,E1 -29844.799,E2 -29844.799} C_VEL
LIN {X 0,Y 62.683,Z 466.971,A -85,B 0,C 180,E1 -29853.762,E2 -29853.762} C_VEL
LIN {X 0,Y 74.8,Z 461.547,A -85,B 0,C 180,E1 -29859.982,E2 -29859.982} C_VEL
LIN {X 0,Y 84.315,Z 456.487,A -85,B 0,C 180,E1 -29863.452,E2 -29863.452} C_VEL
LIN {X 0,Y 95.63,Z 449.5,A -85,B 0,C 180,E1 -29866.611,E2 -29866.611} C_VEL
LIN {X 0,Y 107.315,Z 440.968,A -85,B 0,C 180,E1 -29869.219,E2 -29869.219} C_VEL
LIN {X 0,Y 119.118,Z 430.763,A -85,B 0,C 180,E1 -29871.213,E2 -29871.213} C_VEL
LIN {X 0,Y 129.334,Z 420.321,A -85,B 0,C 180,E1 -29872.618,E2 -29872.618} C_VEL
LIN {X 0,Y 138.754,Z 408.962,A -85,B 0,C 180,E1 -29873.735,E2 -29873.735} C_VEL
LIN {X 0,Y 147.404,Z 396.531,A -85,B 0,C 180,E1 -29874.67,E2 -29874.67} C_VEL
LIN {X 0,Y 155.107,Z 383.118,A -85,B 0,C 180,E1 -29875.442,E2 -29875.442} C_VEL
LIN {X 0,Y 161.599,Z 369.117,A -85,B 0,C 180,E1 -29875.998,E2 -29875.998} C_VEL
LIN {X 0,Y 167.067,Z 353.904,A -85,B 0,C 180,E1 -29876.425,E2 -29876.425} C_VEL
LIN {X 0,Y 170.998,Z 338.829,A -85,B 0,C 180,E1 -29876.746,E2 -29876.746} C_VEL
LIN {X 0,Y 172.826,Z 328.706,A -85,B 0,C 180,E1 -29876.909,E2 -29876.909} C_VEL
LIN {X 0,Y 172.844,Z 326.922,A -85,B 0,C 180,E1 -29880,E2 -29880} C_VEL
LIN {X 0,Y 172.83,Z 328.683,A -85,B 0,C 180,E1 -29882.983,E2 -29882.983} C_VEL
LIN {X 0,Y 169.78,Z 344.07,A -85,B 0,C 180,E1 -29883.262,E2 -29883.262} C_VEL
LIN {X 0,Y 165.339,Z 359.223,A -85,B 0,C 180,E1 -29883.602,E2 -29883.602} C_VEL
LIN {X 0,Y 160.271,Z 372.291,A -85,B 0,C 180,E1 -29883.964,E2 -29883.964} C_VEL
LIN {X 0,Y 153.331,Z 386.505,A -85,B 0,C 180,E1 -29884.492,E2 -29884.492} C_VEL
LIN {X 0,Y 145.561,Z 399.457,A -85,B 0,C 180,E1 -29885.24,E2 -29885.24} C_VEL
LIN {X 0,Y 137.055,Z 411.31,A -85,B 0,C 180,E1 -29886.175,E2 -29886.175} C_VEL
LIN {X 0,Y 127.535,Z 422.504,A -85,B 0,C 180,E1 -29887.287,E2 -29887.287} C_VEL
LIN {X 0,Y 117.304,Z 432.709,A -85,B 0,C 180,E1 -29888.674,E2 -29888.674} C_VEL
LIN {X 0,Y 105.489,Z 442.676,A -85,B 0,C 180,E1 -29890.674,E2 -29890.674} C_VEL
LIN {X 0,Y 92.235,Z 452.028,A -85,B 0,C 180,E1 -29893.708,E2 -29893.708} C_VEL
LIN {X 0,Y 80.888,Z 458.732,A -85,B 0,C 180,E1 -29897.11,E2 -29897.11} C_VEL
LIN {X 0,Y 68.349,Z 464.917,A -85,B 0,C 180,E1 -29902.267,E2 -29902.267} C_VEL
LIN {X 0,Y 56.681,Z 469.701,A -85,B 0,C 180,E1 -29909.779,E2 -29909.779} C_VEL
LIN {X 0,Y 46.342,Z 473.205,A -85,B 0,C 180,E1 -29920.686,E2 -29920.686} C_VEL
LIN {X 0,Y 38.35,Z 475.51,A -85,B 0,C 180,E1 -29936.648,E2 -29936.648} C_VEL
LIN {X 0,Y 34.325,Z 476.669,A -85,B 0,C 180,E1 -29958.185,E2 -29958.185} C_VEL
LIN {X 0,Y 34.079,Z 476.823,A -85,B 0,C 180,E1 -29969.999,E2 -29969.999} C_VEL
LIN {X 0,Y 35.774,Z 476.207,A -85,B 0,C 180,E1 -29993.135,E2 -29993.135} C_VEL
LIN {X 0,Y 41.917,Z 474.447,A -85,B 0,C 180,E1 -30012.118,E2 -30012.118} C_VEL
LIN {X 0,Y 51.261,Z 471.524,A -85,B 0,C 180,E1 -30025.347,E2 -30025.347} C_VEL
LIN {X 0,Y 62.358,Z 467.365,A -85,B 0,C 180,E1 -30034.372,E2 -30034.372} C_VEL
LIN {X 0,Y 74.533,Z 461.862,A -85,B 0,C 180,E1 -30040.551,E2 -30040.551} C_VEL
LIN {X 0,Y 87.345,Z 454.866,A -85,B 0,C 180,E1 -30044.916,E2 -30044.916} C_VEL
LIN {X 0,Y 98.834,Z 447.358,A -85,B 0,C 180,E1 -30047.992,E2 -30047.992} C_VEL
LIN {X 0,Y 110.542,Z 438.362,A -85,B 0,C 180,E1 -30050.215,E2 -30050.215} C_VEL
LIN {X 0,Y 122.398,Z 427.512,A -85,B 0,C 180,E1 -30052.09,E2 -30052.09} C_VEL
LIN {X 0,Y 132.67,Z 416.342,A -85,B 0,C 180,E1 -30053.339,E2 -30053.339} C_VEL
LIN {X 0,Y 142.113,Z 404.093,A -85,B 0,C 180,E1 -30054.414,E2 -30054.414} C_VEL
LIN {X 0,Y 150.736,Z 390.614,A -85,B 0,C 180,E1 -30055.276,E2 -30055.276} C_VEL
LIN {X 0,Y 157.66,Z 377.36,A -85,B 0,C 180,E1 -30055.874,E2 -30055.874} C_VEL
LIN {X 0,Y 163.887,Z 362.453,A -85,B 0,C 180,E1 -30056.34,E2 -30056.34} C_VEL
LIN {X 0,Y 168.735,Z 347.017,A -85,B 0,C 180,E1 -30056.66,E2 -30056.66} C_VEL
LIN {X 0,Y 172.151,Z 331.104,A -85,B 0,C 180,E1 -30056.926,E2 -30056.926} C_VEL
LIN {X 0,Y 172.533,Z 328.42,A -85,B 0,C 180,E1 -30057.015,E2 -30057.015} C_VEL
LIN {X 0,Y 172.555,Z 326.555,A -85,B 0,C 180,E1 -30060,E2 -30060} C_VEL
LIN {X 0,Y 172.477,Z 327.677,A -85,B 0,C 180,E1 -30061.904,E2 -30061.904} C_VEL
LIN {X 0,Y 172.378,Z 328.733,A -85,B 0,C 180,E1 -30062.356,E2 -30062.356} C_VEL
LIN {X 0,Y 172.004,Z 331.341,A -85,B 0,C 180,E1 -30062.587,E2 -30062.587} C_VEL
LIN {X 0,Y 171.334,Z 334.751,A -85,B 0,C 180,E1 -30062.42,E2 -30062.42} C_VEL
LIN {X 0,Y 169.316,Z 343.641,A -85,B 0,C 180,E1 -30061.322,E2 -30061.322} C_VEL
LIN {X 0,Y 168.279,Z 347.583,A -85,B 0,C 180,E1 -30061.098,E2 -30061.098} C_VEL
LIN {X 0,Y 168.048,Z 348.377,A -85,B 0,C 180,E1 -30061.109,E2 -30061.109} C_VEL
LIN {X 0,Y 163.328,Z 363.011,A -85,B 0,C 180,E1 -30061.443,E2 -30061.443} C_VEL
LIN {X 0,Y 157.331,Z 377.194,A -85,B 0,C 180,E1 -30061.823,E2 -30061.823} C_VEL
LIN {X 0,Y 150.348,Z 390.428,A -85,B 0,C 180,E1 -30062.33,E2 -30062.33} C_VEL
LIN {X 0,Y 141.532,Z 404.041,A -85,B 0,C 180,E1 -30063.149,E2 -30063.149} C_VEL
LIN {X 0,Y 132.09,Z 416.103,A -85,B 0,C 180,E1 -30063.96,E2 -30063.96} C_VEL
LIN {X 0,Y 121.703,Z 427.244,A -85,B 0,C 180,E1 -30065.039,E2 -30065.039} C_VEL
LIN {X 0,Y 109.653,Z 438.06,A -85,B 0,C 180,E1 -30066.564,E2 -30066.564} C_VEL
LIN {X 0,Y 98.272,Z 446.646,A -85,B 0,C 180,E1 -30068.392,E2 -30068.392} C_VEL
LIN {X 0,Y 85.937,Z 454.491,A -85,B 0,C 180,E1 -30071.077,E2 -30071.077} C_VEL
LIN {X 0,Y 75.959,Z 459.841,A -85,B 0,C 180,E1 -30073.712,E2 -30073.712} C_VEL
LIN {X 0,Y 63.02,Z 465.678,A -85,B 0,C 180,E1 -30078.574,E2 -30078.574} C_VEL
LIN {X 0,Y 53.717,Z 469.135,A -85,B 0,C 180,E1 -30083.675,E2 -30083.675} C_VEL
LIN {X 0,Y 42.295,Z 472.628,A -85,B 0,C 180,E1 -30093.816,E2 -30093.816} C_VEL
LIN {X 0,Y 32.927,Z 474.932,A -85,B 0,C 180,E1 -30110.185,E2 -30110.185} C_VEL
LIN {X 0,Y 27.562,Z 476.098,A -85,B 0,C 180,E1 -30135.228,E2 -30135.228} C_VEL
LIN {X 0,Y 27.065,Z 476.251,A -85,B 0,C 180,E1 -30150.001,E2 -30150.001} C_VEL
LIN {X 0,Y 29.595,Z 475.682,A -85,B 0,C 180,E1 -30178.356,E2 -30178.356} C_VEL
LIN {X 0,Y 37.196,Z 473.988,A -85,B 0,C 180,E1 -30199.094,E2 -30199.094} C_VEL
LIN {X 0,Y 47.837,Z 471.129,A -85,B 0,C 180,E1 -30211.825,E2 -30211.825} C_VEL
LIN {X 0,Y 59.862,Z 467.037,A -85,B 0,C 180,E1 -30219.923,E2 -30219.923} C_VEL
LIN {X 0,Y 72.662,Z 461.613,A -85,B 0,C 180,E1 -30225.29,E2 -30225.29} C_VEL
LIN {X 0,Y 82.565,Z 456.552,A -85,B 0,C 180,E1 -30228.208,E2 -30228.208} C_VEL
LIN {X 0,Y 94.262,Z 449.541,A -85,B 0,C 180,E1 -30230.877,E2 -30230.877} C_VEL
LIN {X 0,Y 106.211,Z 441.032,A -85,B 0,C 180,E1 -30233.006,E2 -30233.006} C_VEL
LIN {X 0,Y 118.239,Z 430.827,A -85,B 0,C 180,E1 -30234.629,E2 -30234.629} C_VEL
LIN {X 0,Y 128.613,Z 420.385,A -85,B 0,C 180,E1 -30235.761,E2 -30235.761} C_VEL
LIN {X 0,Y 138.159,Z 409.025,A -85,B 0,C 180,E1 -30236.664,E2 -30236.664} C_VEL
LIN {X 0,Y 147.022,Z 396.421,A -85,B 0,C 180,E1 -30237.441,E2 -30237.441} C_VEL
LIN {X 0,Y 154.705,Z 383.179,A -85,B 0,C 180,E1 -30238.067,E2 -30238.067} C_VEL
LIN {X 0,Y 161.26,Z 369.177,A -85,B 0,C 180,E1 -30238.514,E2 -30238.514} C_VEL
LIN {X 0,Y 166.775,Z 353.961,A -85,B 0,C 180,E1 -30238.854,E2 -30238.854} C_VEL
LIN {X 0,Y 170.755,Z 338.823,A -85,B 0,C 180,E1 -30239.116,E2 -30239.116} C_VEL
LIN {X 0,Y 171.586,Z 334.526,A -85,B 0,C 180,E1 -30239.208,E2 -30239.208} C_VEL
LIN {X 0,Y 171.663,Z 334.059,A -85,B 0,C 180,E1 -30240,E2 -30240} C_VEL
LIN {X 0,Y 171.596,Z 334.488,A -85,B 0,C 180,E1 -30240.696,E2 -30240.696} C_VEL
LIN {X 0,Y 168.106,Z 349.373,A -85,B 0,C 180,E1 -30240.956,E2 -30240.956} C_VEL
LIN {X 0,Y 163.431,Z 363.652,A -85,B 0,C 180,E1 -30241.217,E2 -30241.217} C_VEL
LIN {X 0,Y 157.312,Z 377.977,A -85,B 0,C 180,E1 -30241.576,E2 -30241.576} C_VEL
LIN {X 0,Y 150.318,Z 391.093,A -85,B 0,C 180,E1 -30242.025,E2 -30242.025} C_VEL
LIN {X 0,Y 141.599,Z 404.462,A -85,B 0,C 180,E1 -30242.724,E2 -30242.724} C_VEL
LIN {X 0,Y 132.037,Z 416.64,A -85,B 0,C 180,E1 -30243.606,E2 -30243.606} C_VEL
LIN {X 0,Y 121.626,Z 427.76,A -85,B 0,C 180,E1 -30244.604,E2 -30244.604} C_VEL
LIN {X 0,Y 109.549,Z 438.547,A -85,B 0,C 180,E1 -30246.071,E2 -30246.071} C_VEL
LIN {X 0,Y 97.653,Z 447.485,A -85,B 0,C 180,E1 -30247.959,E2 -30247.959} C_VEL
LIN {X 0,Y 85.767,Z 454.993,A -85,B 0,C 180,E1 -30250.478,E2 -30250.478} C_VEL
LIN {X 0,Y 72.464,Z 461.944,A -85,B 0,C 180,E1 -30254.1,E2 -30254.1} C_VEL
LIN {X 0,Y 59.624,Z 467.409,A -85,B 0,C 180,E1 -30259.442,E2 -30259.442} C_VEL
LIN {X 0,Y 47.581,Z 471.541,A -85,B 0,C 180,E1 -30267.596,E2 -30267.596} C_VEL
LIN {X 0,Y 36.943,Z 474.437,A -85,B 0,C 180,E1 -30280.451,E2 -30280.451} C_VEL
LIN {X 0,Y 29.353,Z 476.165,A -85,B 0,C 180,E1 -30301.389,E2 -30301.389} C_VEL
LIN {X 0,Y 26.986,Z 476.756,A -85,B 0,C 180,E1 -30329.999,E2 -30329.999} C_VEL
